CASE stControl.nTargetApplicationMode OF
	E_SEW_MoviC_Position_OperationMode.Jog:
		_bOpModeValid := TRUE;
	E_SEW_MoviC_Position_OperationMode.JogNoEnc:
		_bOpModeValid := TRUE;
	E_SEW_MoviC_Position_OperationMode.SpeedControl:
		_bOpModeValid := TRUE;
	E_SEW_MoviC_Position_OperationMode.ReferenceParam:
		_bOpModeValid := TRUE;
	E_SEW_MoviC_Position_OperationMode.ReferenceBus:
		_bOpModeValid := TRUE;
	E_SEW_MoviC_Position_OperationMode.PositionAbs, E_SEW_MoviC_Position_OperationMode.EnergyOptimized, E_SEW_MoviC_Position_OperationMode.MechanicsOptimized:
		_bOpModeValid := TRUE;
	E_SEW_MoviC_Position_OperationMode.PositionRel:
		_bOpModeValid := TRUE;
	E_SEW_MoviC_Position_OperationMode.PositionModPos:
		_bOpModeValid := TRUE;
	E_SEW_MoviC_Position_OperationMode.PositionModNeg:
		_bOpModeValid := TRUE;
	E_SEW_MoviC_Position_OperationMode.PositionModShort:
		_bOpModeValid := TRUE;
END_CASE

(* Base state of the controller *)
_fbBaseState.bStandstill := OC_Core.F_Compare(_fbBasicDrive.fVelocity, 0, 1E-3);
_fbBaseState.nControl.b0_On := stControl.b1_EnableBusStop AND _fbBaseState.eState <> E_ProfidriveGSM_State.S1_SwitchingOnInhibited;
_fbBaseState.nControl.b1_CoastStop := NOT stControl.b13_ActivateInhibit AND bSTO;
_fbBaseState.nControl.b2_QuickStop := stControl.b0_EnableEStop;
_fbBaseState.nControl.b3_EnableOperation := stControl.b7_StartStop AND _bOpModeValid;

_fbBaseState();
		
(* Set parameter of basic drive *)
IF stControl.b12_DisableSoftwareLimits THEN
	_fbBasicDrive.fPositionLimitMin := -2147483648.0;
	_fbBasicDrive.fPositionLimitMax := 2147483647.0;
	_fbBasicDrive.fTolerance := 0.1;
ELSE
	_fbBasicDrive.fPositionLimitMin := DINT_TO_REAL(stConfig.nSoftwareLimitMin);
	_fbBasicDrive.fPositionLimitMax := DINT_TO_REAL(stConfig.nSoftwareLimitMax);
	_fbBasicDrive.fTolerance := 0.1;
END_IF
					
(* Evaluate base state *)
CASE _fbBaseState.eState OF
	
(* S1, S2 or S3 -> Drive coasts to a stop or brake is applied *)
	E_ProfidriveGSM_State.S1_SwitchingOnInhibited,
	E_ProfidriveGSM_State.S2_ReadyForSwitchingOn,
	E_ProfidriveGSM_State.S3_SwitchedOn:
		_fbBasicDrive.Stop(stConfig.fDecCoastStop);

(* S4 -> Evaluate operation mode *)
	E_ProfidriveGSM_State.S4_Operation:
		Operation();

(* S5a -> Drive decelerates with application limit *)
	E_ProfidriveGSM_State.S51_RampStop:
		_fbBasicDrive.Stop(stConfig.fDecelerationLimit);
		
(* S5b -> Drive decelerates with emergency stop ramp *)
	E_ProfidriveGSM_State.S52_QuickStop:
	    _fbBasicDrive.Stop(stConfig.fDecEstop);
END_CASE
	
(* Status Word *)
stStatus.b0_InverterReady				:= TRUE;
stStatus.b1_STOInactive					:= bSTO;
stStatus.b2_PowerStageOn				:= stControl.b13_ActivateInhibit;
stStatus.b3_BrakeReleased				:= stControl.b1_EnableBusStop OR stControl.b3_ReleaseBrake;
stStatus.b4_MotorTurning				:= NOT _fbBaseState.bStandstill;
stStatus.b5_DriveReferenced				:= TRUE;
stStatus.b6_SetpointsActive		 		:= FALSE;
stStatus.b7_TargetpositionReached		:= _fbBasicDrive.bIsPositionReached;	
stStatus.b8_ErrorActive					:= FALSE;
stStatus.b9_WarningActive				:= FALSE;
stStatus.b10_DriveTrain2Active			:= stControl.b10_ActivateDriveTrain2;
stStatus.b11_SpeedSetpointReached		:= _fbBasicDrive.bIsMoving;
stStatus.b12_SoftwareLimitsDisabled		:= stControl.b12_DisableSoftwareLimits;
stStatus.b13_OutputStageInhibit			:= _fbBaseState.nStatus.b6_SwitchingOnInhibited;
stStatus.b14_StandByModeActive			:= stControl.b14_ActivateStandByMode;
stStatus.b15_MovikitHeartbeat			:= stControl.b15_MovikitHeartbeat;

(* Status values *)
stStatus.nActualSpeed := REAL_TO_INT(_fbBasicDrive.fVelocity / stConfig.fRatioVelocity);
stStatus.nActualStatus := 0;
stStatus.nActualTorque := 0;
stStatus.nDigitalInputs := nDigitalInputs;
IF _bOpModeValid THEN
	stStatus.nActualApplicationMode := stControl.nTargetApplicationMode;
END_IF
stStatus.nActualPosition := REAL_TO_DINT(_fbBasicDrive.fPosition);
	
(* Position output *)
THIS^.ControlData := _fbBasicDrive.fPosition * stConfig.fRatioPosition + stConfig.fPositionOffset;
fValue := ControlData;
END_METHOD

METHOD INTERNAL GetControlData : BOOL
IF pControl <= 0 OR stConfig.bForceMode THEN RETURN; END_IF

(* PO1 Control Word *)
F_Memcpy(ADR(stControl), pControl, 2, stConfig.bSwapProcessData);
(* PO2 Setpoint Speed *)
F_Memcpy(ADR(stControl) + 2, pControl + 2, 2, stConfig.bSwapProcessData);
(* PO3 Setpoint Acceleration *)
F_Memcpy(ADR(stControl) + 4, pControl + 4, 2, stConfig.bSwapProcessData);
(* PO4 Setpoint Deceleration *)
F_Memcpy(ADR(stControl) + 6, pControl + 6, 2, stConfig.bSwapProcessData);
(* PO5 Digital Outputs *)
F_Memcpy(ADR(stControl) + 8, pControl + 8, 2, stConfig.bSwapProcessData);
(* PO6 Target Application Mode *)
F_Memcpy(ADR(stControl) + 10, pControl + 10, 2, stConfig.bSwapProcessData);
(* PO7,PO8 Target Position *)
F_Memcpy(ADR(stControl) + 12, pControl + 12, 4, stConfig.bSwapProcessData);
END_METHOD

METHOD INTERNAL InitRun
VAR_INST
	bInitRun : BOOL := TRUE;
END_VAR
IF NOT bInitRun THEN RETURN; END_IF
bInitRun := FALSE;

IF pControl = 0 OR pStatus = 0 THEN
	ADSLOGSTR(ADSLOG_MSGTYPE_WARN, CONCAT(_sPath, ': %s'), 'Plc address not set.');
END_IF

_fbBasicDrive.fPosition := stConfig.fInitPosition;
END_METHOD

METHOD PRIVATE Operation
VAR_INST
	fTargetPos			: REAL;
	fSetpointVel		: REAL;
	fSetpointAcc		: REAL;
	fSetpointDec		: REAL;
END_VAR
(* Copy setpoint values *)
fTargetPos 		:= DINT_TO_REAL(stControl.nTargetPosition);
fSetpointVel 	:= stControl.nSetpointSpeed * stConfig.fRatioVelocity; 
fSetpointAcc 	:= stControl.nSetpointAcceleration * stConfig.fRatioAccDec;
fSetpointDec 	:= stControl.nSetpointDeceleration * stConfig.fRatioAccDec;

(* Operation statemachine *)
CASE stStatus.nActualApplicationMode OF	
	E_SEW_MoviC_Position_OperationMode.Jog:
		IF stControl.b4_JoggingCW AND NOT stControl.b5_JoggingCCW THEN
			_fbBasicDrive.MoveAbsolute(DINT_TO_REAL(stConfig.nSoftwareLimitMax), fSetpointVel, fSetpointAcc, fSetpointDec);
		ELSIF stControl.b5_JoggingCCW AND NOT stControl.b4_JoggingCW THEN
			_fbBasicDrive.MoveAbsolute(DINT_TO_REAL(stConfig.nSoftwareLimitMin), fSetpointVel, fSetpointAcc, fSetpointDec);
		ELSE
			_fbBasicDrive.Stop(fSetpointDec);
		END_IF
		
	E_SEW_MoviC_Position_OperationMode.JogNoEnc:			
		IF stControl.b4_JoggingCW AND NOT stControl.b5_JoggingCCW THEN
			_fbBasicDrive.MoveVelocity(fSetpointVel, fSetpointAcc, fSetpointDec);
		ELSIF stControl.b5_JoggingCCW AND NOT stControl.b4_JoggingCW THEN
			_fbBasicDrive.MoveVelocity(-fSetpointVel, fSetpointAcc, fSetpointDec);
		ELSE
			_fbBasicDrive.Stop(fSetpointDec);
		END_IF
		
	E_SEW_MoviC_Position_OperationMode.SpeedControl:
		_fbBasicDrive.MoveVelocity(fSetpointVel, fSetpointAcc, fSetpointDec);
	
	E_SEW_MoviC_Position_OperationMode.ReferenceParam:
		//not yet implemented
		
	E_SEW_MoviC_Position_OperationMode.ReferenceBus:
		//not yet implemented
	
	E_SEW_MoviC_Position_OperationMode.PositionAbs, E_SEW_MoviC_Position_OperationMode.EnergyOptimized, E_SEW_MoviC_Position_OperationMode.MechanicsOptimized:
		IF stControl.b7_StartStop THEN						
			_fbBasicDrive.MoveAbsolute(fTargetPos, fSetpointVel, fSetpointAcc, fSetpointDec);
		ELSE
			_fbBasicDrive.Stop(fSetpointDec);
		END_IF
	
	E_SEW_MoviC_Position_OperationMode.PositionRel:
		//not yet implemented
		
	E_SEW_MoviC_Position_OperationMode.PositionModPos:
		//not yet implemented
		
	E_SEW_MoviC_Position_OperationMode.PositionModNeg:
		//not yet implemented
		
	E_SEW_MoviC_Position_OperationMode.PositionModShort:
		//not yet implemented
END_CASE
END_METHOD

METHOD INTERNAL Safety
VAR_INPUT
END_VAR
(* Check if Movisafe is available *)
IF iMovisafe <> 0 THEN
	bSTO := iMovisafe.bSTO;
END_IF
END_METHOD

METHOD INTERNAL SetStatusData
IF pStatus <= 0 THEN RETURN; END_IF

(* PI1 Status Word *)
F_Memcpy(pStatus, ADR(stStatus), 2, stConfig.bSwapProcessData);
(* PI2 Actual Speed *)
F_Memcpy(pStatus + 2, ADR(stStatus) + 2, 2, stConfig.bSwapProcessData);
(* PI3 Actual Status *)
F_Memcpy(pStatus + 4, ADR(stStatus) + 4, 2, stConfig.bSwapProcessData);
(* PI4 Actual Torque *)
F_Memcpy(pStatus + 6, ADR(stStatus) + 6, 2, stConfig.bSwapProcessData);
(* PI5 Digital Inputs *)
F_Memcpy(pStatus + 8, ADR(stStatus) + 8, 2, stConfig.bSwapProcessData);
(* PI6 Actual Application Mode *)
F_Memcpy(pStatus + 10, ADR(stStatus) + 10, 2, stConfig.bSwapProcessData);
(* PI7,PI8 Actual Position *)
F_Memcpy(pStatus + 12, ADR(stStatus) + 12, 4, stConfig.bSwapProcessData);
END_METHOD

END_FUNCTION_BLOCK

// ---- Tests/Helpers/FB_SEW_Movisafe.TcPOU
FUNCTION_BLOCK FB_SEW_Movisafe IMPLEMENTS I_SEW_Movisafe
VAR_INPUT
	bSetSTO : BOOL;
END_VAR
VAR_OUTPUT
END_VAR
VAR
END_VAR

PROPERTY bSTO : BOOL
GET
bSTO := bSetSTO;
END_GET
END_PROPERTY

END_FUNCTION_BLOCK

// ---- Tests/Devices/FB_SEW_MoviC_Velocity_Test.TcPOU
FUNCTION_BLOCK FB_SEW_MoviC_Velocity_Test EXTENDS TcUnit.FB_TestSuite

Test_ProcessDataControl();
Test_ProcessDataStatus();
Test_Safety();
Test_Cycle_Status_Const_Mirror();
Test_Cycle_Status_Movement('Test Movement 0',0,1,FALSE,FALSE );
Test_Cycle_Status_Movement('Test Movement 1000, Gear 1',1000,1,TRUE,TRUE );
Test_Cycle_Status_Movement('Test Movement -5000, Gear 1',-5000,1,TRUE,TRUE );
Test_Cycle_Status_Movement('Test Movement 1000, Gear 5',1000,5,TRUE,TRUE );
Test_Cycle_Status_Movement('Test Movement 1000, Gear -0,5',1000,-0.5,TRUE,TRUE );

METHOD Test_Cycle_Status_Const_Mirror : REFERENCE TO FB_Test
VAR
	fbDrive 			: FB_SEW_MoviC_Velocity;
	bExpected			: BOOL;
	nIntExpected		: INT;
	nWordExpected		: WORD;
	stExpected			: ST_SEW_MoviC_Velocity_Status;
	bResult 			: BOOL;	
	nIntResult 			: INT;	
	nWordResult 		: WORD;	
	stResult			: ST_SEW_MoviC_Velocity_Status;
	
	stSetControl		: ST_SEW_MoviC_Velocity_Control;
END_VAR
TEST('Status CONST TRUE');

bExpected := TRUE;

fbDrive.Cycle();

stResult := fbDrive.stStatus;

bResult := BIT_TO_BOOL(stResult.b0_InverterReady);

AssertEquals(Expected := bExpected,
             Actual := bResult,
             Message := 'InverterReady not set correctly');

bResult := BIT_TO_BOOL(stResult.b5_DriveReferenced);
			 
AssertEquals(Expected := bExpected,
             Actual := bResult,
             Message := 'DriveReferenced not set correctly');
			 
bResult := BIT_TO_BOOL(stResult.b2_PowerStageOn);
			 
AssertEquals(Expected := bExpected,
             Actual := bResult,
             Message := 'PowerStageOn not set correctly');
	 
TEST_FINISHED();

TEST('Status CONST FALSE');

bExpected := FALSE;

fbDrive.Cycle();

stResult := fbDrive.stStatus;

bResult := BIT_TO_BOOL(stResult.b6_SetpointsActive);

AssertEquals(Expected := bExpected,
             Actual := bResult,
             Message := 'SetpointsActive not set correctly');
			 
bResult := BIT_TO_BOOL(stResult.b7_TargetpositionReached);

AssertEquals(Expected := bExpected,
             Actual := bResult,
             Message := 'TargetpositionReached not set correctly');

bResult := BIT_TO_BOOL(stResult.b8_ErrorActive);
			 
AssertEquals(Expected := bExpected,
             Actual := bResult,
             Message := 'ErrorActive not set correctly');

bResult := BIT_TO_BOOL(stResult.b9_WarningActive);
			 
AssertEquals(Expected := bExpected,
             Actual := bResult,
             Message := 'WarningActive not set correctly');
	 
TEST_FINISHED();

TEST('Status CONST 0');

nWordExpected := 0;
nIntExpected := 0;

fbDrive.Cycle();

stResult := fbDrive.stStatus;

nWordResult := stResult.nActualStatus;

AssertEquals(Expected := nWordExpected,
             Actual := nWordResult,
             Message := 'ActualStatus not set correctly');

nIntResult := stResult.nActualTorque;
			 
AssertEquals(Expected := nIntExpected,
             Actual := nIntResult,
             Message := 'ActualTorque not set correctly');
			 
nWordResult := stResult.nDigitalInputs;

AssertEquals(Expected := nWordExpected,
             Actual := nWordResult,
             Message := 'DigitalInputs not set correctly');
	 
TEST_FINISHED();


TEST('Status Mirror Control FALSE');

bExpected := FALSE;

stSetControl.b13_ActivateInhibit := bExpected;
stSetControl.b10_ActivateDriveTrain2 := bExpected;
stSetControl.b12_DisableSoftwareLimits := bExpected;
stSetControl.b14_ActivateStandByMode := bExpected;
stSetControl.b15_MovikitHeartbeat := bExpected;

fbDrive.stControl := stSetControl;

fbDrive.Cycle();

stResult := fbDrive.stStatus;

bResult := BIT_TO_BOOL(stResult.b10_DriveTrain2Active);
			 
AssertEquals(Expected := bExpected,
             Actual := bResult,
             Message := 'riveTrain2Active not set correctly');

bResult := BIT_TO_BOOL(stResult.b12_SoftwareLimitsDisabled);
			 
AssertEquals(Expected := bExpected,
             Actual := bResult,
             Message := 'SoftwareLimitsDisabled not set correctly');
			 
 bResult := BIT_TO_BOOL(stResult.b14_StandByModeActive);
			 
AssertEquals(Expected := bExpected,
             Actual := bResult,
             Message := 'StandByModeActive not set correctly');
			 
bResult := BIT_TO_BOOL(stResult.b15_MovikitHeartbeat);
			 
AssertEquals(Expected := bExpected,
             Actual := bResult,
             Message := 'MovikitHeartbeat not set correctly');
	 
TEST_FINISHED();

TEST('Status Mirror Control TRUE');

bExpected := TRUE;

stSetControl.b13_ActivateInhibit := bExpected;
stSetControl.b10_ActivateDriveTrain2 := bExpected;
stSetControl.b12_DisableSoftwareLimits := bExpected;
stSetControl.b14_ActivateStandByMode := bExpected;
stSetControl.b15_MovikitHeartbeat := bExpected;

fbDrive.stControl := stSetControl;

fbDrive.Cycle();

stResult := fbDrive.stStatus;

bResult := BIT_TO_BOOL(stResult.b10_DriveTrain2Active);
			 
AssertEquals(Expected := bExpected,
             Actual := bResult,
             Message := 'DriveTrain2Active not set correctly');

bResult := BIT_TO_BOOL(stResult.b12_SoftwareLimitsDisabled);
			 
AssertEquals(Expected := bExpected,
             Actual := bResult,
             Message := 'SoftwareLimitsDisabled not set correctly');
			 
 bResult := BIT_TO_BOOL(stResult.b14_StandByModeActive);
			 
AssertEquals(Expected := bExpected,
             Actual := bResult,
             Message := 'StandByModeActive not set correctly');
			 
bResult := BIT_TO_BOOL(stResult.b15_MovikitHeartbeat);
			 
AssertEquals(Expected := bExpected,
             Actual := bResult,
             Message := 'MovikitHeartbeat not set correctly');
	 
TEST_FINISHED();
END_METHOD

METHOD Test_Cycle_Status_Movement : REFERENCE TO FB_Test
VAR_INPUT
	sName 								: T_MaxString;
	nVelcity							: INT;
	fRatioVelcity						: REAL;
	bExpected_b4_MotorTurning 			: BOOL;
	bExpected_b11_SpeedSetpointReached 	: BOOL;
END_VAR
VAR
	nCycle		: INT;
	fbDrive 	: FB_SEW_MoviC_Velocity;
	bResult		: BOOL;	
	nResult 	: INT;
END_VAR
TEST(sName);

// Start Conditions
fbDrive.stControl.b0_EnableEStop := TRUE;
fbDrive.stControl.b1_EnableBusStop := TRUE;
fbDrive.stControl.b7_StartStop := TRUE;
fbDrive.stControl.b13_ActivateInhibit := FALSE;
fbDrive.bSTO := TRUE;
fbDrive.stControl.nSetpointSpeed := nVelcity;
fbDrive.stControl.nSetpointAcceleration := 1000;
fbDrive.stControl.nSetpointDeceleration := 1000;

fbDrive.stConfig.fRatioPosition := fRatioVelcity;

FOR nCycle := 1 TO 5500 DO
	fbDrive.Cycle();
END_FOR

nResult := fbDrive.stStatus.nActualSpeed;

AssertEquals(Expected := nVelcity,
             Actual := nResult,
             Message := 'ActualSpeed not set correctly');

bResult := fbDrive.stStatus.b4_MotorTurning;

AssertEquals(Expected := bExpected_b4_MotorTurning,
             Actual := bResult,
             Message := 'b4_MotorTurning not set correctly');


bResult := fbDrive.stStatus.b11_SpeedSetpointReached;
			 
AssertEquals(Expected := bExpected_b11_SpeedSetpointReached,
             Actual := bResult,
             Message := 'b11_SpeedSetpointReached not set correctly');
	 
TEST_FINISHED();
END_METHOD

METHOD Test_ProcessDataControl : REFERENCE TO FB_Test
VAR
	fbDrive 						: FB_SEW_MoviC_Velocity;
	
	nExpectedCW						: WORD;
	nExpectedSetpointSpeed			: INT;
	nExpectedSetpointAcceleration	: INT;
	nExpectedSetpointDeceleration	: INT;
	nExpectedDigitalOutputs			: WORD;
	
	nActualCW						: WORD;
	nActualSetpointSpeed			: INT;
	nActualSetpointAcceleration		: INT;
	nActualSetpointDeceleration		: INT;
	nActualDigitalOutputs			: WORD;
		
	stExpectedControlData 			: ST_SEW_MoviC_Velocity_Control;		
	stActualControlData				: ST_SEW_MoviC_Velocity_Control;	
END_VAR
TEST('Process data to control structure');

//Arrange
nExpectedCW := 16#A1B2;					
nExpectedSetpointSpeed := UINT_TO_INT(16#C3D4);		
nExpectedSetpointAcceleration := UINT_TO_INT(16#E5F6);		
nExpectedSetpointDeceleration := UINT_TO_INT(16#B6A5);	
nExpectedDigitalOutputs := 16#D4C3;			

F_Memcpy(ADR(stExpectedControlData), ADR(nExpectedCW), 2, FALSE);
F_Memcpy(ADR(stExpectedControlData) + 2, ADR(nExpectedSetpointSpeed), 2, FALSE);
F_Memcpy(ADR(stExpectedControlData) + 4, ADR(nExpectedSetpointAcceleration), 2, FALSE);
F_Memcpy(ADR(stExpectedControlData) + 6, ADR(nExpectedSetpointDeceleration), 2, FALSE);
F_Memcpy(ADR(stExpectedControlData) + 8, ADR(nExpectedDigitalOutputs), 2, FALSE);

fbDrive.pControl := ADR(stExpectedControlData);

//Act
fbDrive.GetControlData();

stActualControlData := fbDrive.stControl;

//Assert
F_Memcpy(ADR(nActualCW), ADR(fbDrive.stControl), 2, FALSE);
//F_Memcpy(ADR(nActualTargetVelocity), ADR(fbDrive.stControl) + 2, 2, FALSE);

AssertEquals(Expected := nExpectedCW,
             Actual := nActualCW,
             Message := 'CW is not correct');
	 
AssertEquals(Expected := nExpectedSetpointSpeed,
             Actual := stActualControlData.nSetpointSpeed,
             Message := 'SetpointSpeed is not correct');
			 
AssertEquals(Expected := nExpectedSetpointAcceleration,
             Actual := stActualControlData.nSetpointAcceleration,
             Message := 'SetpointAcceleration is not correct');
			 
AssertEquals(Expected := nExpectedSetpointDeceleration,
             Actual := stActualControlData.nSetpointDeceleration,
             Message := 'SetpointSpeed is not correct');
			 
AssertEquals(Expected := nExpectedDigitalOutputs,
             Actual := stActualControlData.nDigitalOutputs,
             Message := 'SetpointDeceleration is not correct');
			 
TEST_FINISHED();


TEST('Process data to control structure SWAP');

//Arrange
F_Memcpy(ADR(stExpectedControlData), ADR(nExpectedCW), 2, TRUE);
F_Memcpy(ADR(stExpectedControlData) + 2, ADR(nExpectedSetpointSpeed), 2, TRUE);
F_Memcpy(ADR(stExpectedControlData) + 4, ADR(nExpectedSetpointAcceleration), 2, TRUE);
F_Memcpy(ADR(stExpectedControlData) + 6, ADR(nExpectedSetpointDeceleration), 2, TRUE);
F_Memcpy(ADR(stExpectedControlData) + 8, ADR(nExpectedDigitalOutputs), 2, TRUE);

fbDrive.stConfig.bSwapProcessData := TRUE;

fbDrive.pControl := ADR(stExpectedControlData);

//Act
fbDrive.GetControlData();

stActualControlData := fbDrive.stControl;

//Assert
AssertEquals(Expected := nExpectedCW,
             Actual := nActualCW,
             Message := 'CW is not correct');
	 
AssertEquals(Expected := nExpectedSetpointSpeed,
             Actual := stActualControlData.nSetpointSpeed,
             Message := 'SetpointSpeed is not correct');
			 
AssertEquals(Expected := nExpectedSetpointAcceleration,
             Actual := stActualControlData.nSetpointAcceleration,
             Message := 'SetpointAcceleration is not correct');
			 
AssertEquals(Expected := nExpectedSetpointDeceleration,
             Actual := stActualControlData.nSetpointDeceleration,
             Message := 'SetpointSpeed is not correct');
			 
AssertEquals(Expected := nExpectedDigitalOutputs,
             Actual := stActualControlData.nDigitalOutputs,
             Message := 'SetpointDeceleration is not correct');

TEST_FINISHED();
END_METHOD

METHOD Test_ProcessDataStatus : REFERENCE TO FB_Test
VAR
	fbDrive 						: FB_SEW_MoviC_Velocity;
	
	nExpectedSW						: WORD;
	nExpectedActualSpeed			: INT;
	nExpectedActualStatus			: WORD;
	nExpectedActualTorque			: INT;
	nExpectedDigitalInputs			: WORD;
	
	nActualSW						: WORD;
	nActualActualSpeed				: INT;
	nActualActualStatus				: WORD;
	nActualActualTorque				: INT;
	nActualDigitalInputs			: WORD;

	stExpectedStatusData 			: ST_SEW_MoviC_Velocity_Status;		
	stActualStatusData 				: ST_SEW_MoviC_Velocity_Status;	
END_VAR
TEST('Assign status structure to process data');

//Arrange
nExpectedSW := 16#A1B2;					
nExpectedActualSpeed := UINT_TO_INT(16#C3D4);		
nExpectedActualStatus := 16#E5F6;		
nExpectedActualTorque := UINT_TO_INT(16#B6A5);	
nExpectedDigitalInputs := 16#B6A5;			
	
F_Memcpy(ADR(fbDrive.stStatus), ADR(nExpectedSW), 2, FALSE);
F_Memcpy(ADR(fbDrive.stStatus) + 2, ADR(nExpectedActualSpeed), 2, FALSE);
F_Memcpy(ADR(fbDrive.stStatus) + 4, ADR(nExpectedActualStatus), 2, FALSE);
F_Memcpy(ADR(fbDrive.stStatus) + 6, ADR(nExpectedActualTorque), 2, FALSE);
F_Memcpy(ADR(fbDrive.stStatus) + 8, ADR(nExpectedDigitalInputs), 2, FALSE);

fbDrive.pStatus := ADR(stActualStatusData);

//Act
fbDrive.SetStatusData();

//Assert
F_Memcpy(ADR(nActualSW), ADR(stActualStatusData), 2, FALSE);
F_Memcpy(ADR(nActualActualSpeed), ADR(stActualStatusData) + 2, 2, FALSE);
F_Memcpy(ADR(nActualActualStatus), ADR(stActualStatusData) + 4, 2, FALSE);
F_Memcpy(ADR(nActualActualTorque), ADR(stActualStatusData) + 6, 2, FALSE);
F_Memcpy(ADR(nActualDigitalInputs), ADR(stActualStatusData) + 8, 2, FALSE);

AssertEquals(Expected := nExpectedSW,
             Actual := nActualSW,
             Message := 'ZSW1 is not correct');
	 
AssertEquals(Expected := nExpectedActualSpeed,
             Actual := nActualActualSpeed,
             Message := 'ActualVelocity is not correct');	

AssertEquals(Expected := nExpectedActualStatus,
             Actual := nActualActualStatus,
             Message := 'ActualVelocity is not correct');

AssertEquals(Expected := nExpectedActualTorque,
             Actual := nActualActualTorque,
             Message := 'ActualVelocity is not correct');	
				 
AssertEquals(Expected := nExpectedDigitalInputs,
             Actual := nActualDigitalInputs,
             Message := 'ActualVelocity is not correct');	
					 			 
TEST_FINISHED();

TEST('Assign status structure to process data SWAP');

//Arrange
nExpectedSW := 16#A1B2;					
nExpectedActualSpeed := UINT_TO_INT(16#C3D4);		
nExpectedActualStatus := 16#E5F6;		
nExpectedActualTorque := UINT_TO_INT(16#B6A5);	
nExpectedDigitalInputs := 16#B6A5;			
	
F_Memcpy(ADR(fbDrive.stStatus), ADR(nExpectedSW), 2, TRUE);
F_Memcpy(ADR(fbDrive.stStatus) + 2, ADR(nExpectedActualSpeed), 2, TRUE);
F_Memcpy(ADR(fbDrive.stStatus) + 4, ADR(nExpectedActualStatus), 2, TRUE);
F_Memcpy(ADR(fbDrive.stStatus) + 6, ADR(nExpectedActualTorque), 2, TRUE);
F_Memcpy(ADR(fbDrive.stStatus) + 8, ADR(nExpectedDigitalInputs), 2, TRUE);

fbDrive.stConfig.bSwapProcessData := TRUE;

fbDrive.pStatus := ADR(stActualStatusData);

//Act
fbDrive.SetStatusData();

//Assert
F_Memcpy(ADR(nActualSW), ADR(stActualStatusData), 2, FALSE);
F_Memcpy(ADR(nActualActualSpeed), ADR(stActualStatusData) + 2, 2, FALSE);
F_Memcpy(ADR(nActualActualStatus), ADR(stActualStatusData) + 4, 2, FALSE);
F_Memcpy(ADR(nActualActualTorque), ADR(stActualStatusData) + 6, 2, FALSE);
F_Memcpy(ADR(nActualDigitalInputs), ADR(stActualStatusData) + 8, 2, FALSE);

AssertEquals(Expected := nExpectedSW,
             Actual := nActualSW,
             Message := 'ZSW1 is not correct');
	 
AssertEquals(Expected := nExpectedActualSpeed,
             Actual := nActualActualSpeed,
             Message := 'ActualVelocity is not correct');	

AssertEquals(Expected := nExpectedActualStatus,
             Actual := nActualActualStatus,
             Message := 'ActualVelocity is not correct');

AssertEquals(Expected := nExpectedActualTorque,
             Actual := nActualActualTorque,
             Message := 'ActualVelocity is not correct');	
				 
AssertEquals(Expected := nExpectedDigitalInputs,
             Actual := nActualDigitalInputs,
             Message := 'ActualVelocity is not correct');			 
			 
TEST_FINISHED();
END_METHOD

METHOD Test_Safety : REFERENCE TO FB_Test
VAR
	fbDrive 					: FB_SEW_MoviC_Velocity;
		
	fbSafe						: FB_SEW_Movisafe;
	
	stExpectedSTO				: BOOL;		
	stActualSTO					: BOOL;	
END_VAR
TEST(' Without Safety Interface STO TRUE');

//Arrange
stExpectedSTO := TRUE;
fbDrive.bSTO := stExpectedSTO;

//Act
fbDrive.Safety();

//Assert
stActualSTO := fbDrive.bSTO;

AssertEquals(Expected := stExpectedSTO,
             Actual := stActualSTO,
             Message := 'STO is not correct');
	 		 
TEST_FINISHED();

TEST(' Without Safety Interface STO FALSE');

//Arrange
stExpectedSTO := FALSE;
fbDrive.bSTO := stExpectedSTO;

//Act
fbDrive.Safety();

//Assert
stActualSTO := fbDrive.bSTO;

AssertEquals(Expected := stExpectedSTO,
             Actual := stActualSTO,
             Message := 'STO is not correct');
	 		 
TEST_FINISHED();

TEST('Safety Interface STO TRUE');

//Arrange
stExpectedSTO := TRUE;

fbSafe.bSetSTO := stExpectedSTO;
fbDrive.iMovisafe := fbSafe;

//Act
fbDrive.Safety();

//Assert
stActualSTO := fbDrive.bSTO;

AssertEquals(Expected := stExpectedSTO,
             Actual := stActualSTO,
             Message := 'STO is not correct');
	 		 
TEST_FINISHED();

TEST('Safety Interface FALSE');

//Arrange
stExpectedSTO := FALSE;

fbSafe.bSetSTO := stExpectedSTO;
fbDrive.iMovisafe := fbSafe;

//Act
fbDrive.Safety();

//Assert
stActualSTO := fbDrive.bSTO;

AssertEquals(Expected := stExpectedSTO,
             Actual := stActualSTO,
             Message := 'STO is not correct');
	 		 
TEST_FINISHED();

TEST('Safety Interface false, Overwrite FB input');

//Arrange
stExpectedSTO := FALSE;

fbSafe.bSetSTO := stExpectedSTO;
fbDrive.iMovisafe := fbSafe;
fbDrive.bSTO := NOT stExpectedSTO;

//Act
fbDrive.Safety();

//Assert
stActualSTO := fbDrive.bSTO;

AssertEquals(Expected := stExpectedSTO,
             Actual := stActualSTO,
             Message := 'STO is not correct');
	 		 
TEST_FINISHED();

TEST('Safety Interface true, Overwrite FB input');

//Arrange
stExpectedSTO := TRUE;

fbSafe.bSetSTO := stExpectedSTO;
fbDrive.iMovisafe := fbSafe;
fbDrive.bSTO := NOT stExpectedSTO;

//Act
fbDrive.Safety();

//Assert
stActualSTO := fbDrive.bSTO;

AssertEquals(Expected := stExpectedSTO,
             Actual := stActualSTO,
             Message := 'STO is not correct');
	 		 
TEST_FINISHED();
END_METHOD

END_FUNCTION_BLOCK

// ---- Devices/SEW_MoviC_Velocity/FB_SEW_MoviC_Velocity.TcPOU
(*
FB_SEW_MoviC_Velocity simulates the funcitionalty of a SEW‑EURODRIVE MOVI-C® CONTROLLER with MOVIKIT® Velocity module.

Disclaimer: This simulation is an independent project and is not affiliated with, endorsed by, or approved by SEW‑EURODRIVE. All rights to the SEW‑EURODRIVE brand name and trademarks remain the property of the manufacturer.
Furthermore, no guarantee is given for the completeness of the functional scope or the error-free operation of the simulation. Users should be aware that deviations from the actual product may occur.
*)

{attribute 'reflection'}
FUNCTION_BLOCK FB_SEW_MoviC_Velocity EXTENDS FB_LinkDataReal

VAR_INPUT
	pControl 			: PVOID; //Pocess data from fieldbus. Size must be >= stControl.
	pStatus 			: PVOID; //Pocess data to fieldbus. Size must be >= stStatus.
	stControl 			: ST_SEW_MoviC_Velocity_Control; //Control structure. Is read from the fieldbus.
	stConfig 			: ST_SEW_MoviC_Velocity_Config; //Config structure. Contains parameters of the device.	
	
	bSTO				: BOOL := TRUE;
	iMovisafe			: I_SEW_Movisafe;
END_VAR

VAR_OUTPUT
	stStatus			: ST_SEW_MoviC_Velocity_Status;
	fValue				: REAL;
END_VAR

VAR
    {attribute 'instance-path'} 
    {attribute 'noinit'} 
    _sPath 				: STRING; 	                			
	                			
	_fbBaseState		: FB_ProfidriveGSM;
	_fbBasicDrive		: FB_DriveControl;	                						
END_VAR

SUPER^();
InitRun();

GetControlData();
Safety();
Cycle();
SetStatusData();

METHOD INTERNAL Cycle
(* Base state of the controller *)
_fbBaseState.bStandstill := OC_Core.F_Compare(_fbBasicDrive.fVelocity, 0, 1E-3);
_fbBaseState.nControl.b0_On := stControl.b1_EnableBusStop AND _fbBaseState.eState <> E_ProfidriveGSM_State.S1_SwitchingOnInhibited;
_fbBaseState.nControl.b1_CoastStop := NOT stControl.b13_ActivateInhibit AND bSTO;
_fbBaseState.nControl.b2_QuickStop := stControl.b0_EnableEStop;
_fbBaseState.nControl.b3_EnableOperation := stControl.b7_StartStop;

_fbBaseState();
					
(* Evaluate base state *)
CASE _fbBaseState.eState OF	
(* S1, S2 or S3 -> Drive coasts to a stop or brake is applied *)
	E_ProfidriveGSM_State.S1_SwitchingOnInhibited,
	E_ProfidriveGSM_State.S2_ReadyForSwitchingOn,
	E_ProfidriveGSM_State.S3_SwitchedOn:
		_fbBasicDrive.Stop(stConfig.fDecCoastStop);

(* S4 -> Operation mode *)
	E_ProfidriveGSM_State.S4_Operation:
		Operation();

(* S5a -> Drive decelerates with application limit *)
	E_ProfidriveGSM_State.S51_RampStop:
		_fbBasicDrive.Stop(stConfig.fDecelerationLimit);
		
(* S5b -> Drive decelerates with emergency stop ramp *)
	E_ProfidriveGSM_State.S52_QuickStop:
	    _fbBasicDrive.Stop(stConfig.fDecEstop);
END_CASE
	
(* Status Word *)
stStatus.b0_InverterReady				:= TRUE;
stStatus.b1_STOInactive					:= bSTO;
stStatus.b2_PowerStageOn				:= _fbBaseState.bPowerOn;
stStatus.b3_BrakeReleased				:= stControl.b1_EnableBusStop OR stControl.b3_ReleaseBrake;
stStatus.b4_MotorTurning				:= NOT _fbBaseState.bStandstill;
stStatus.b5_DriveReferenced				:= TRUE;
stStatus.b6_SetpointsActive		 		:= FALSE;
stStatus.b7_TargetpositionReached		:= FALSE;	
stStatus.b8_ErrorActive					:= FALSE;
stStatus.b9_WarningActive				:= FALSE;
stStatus.b10_DriveTrain2Active			:= stControl.b10_ActivateDriveTrain2;
stStatus.b11_SpeedSetpointReached		:= _fbBasicDrive.bIsMoving;
stStatus.b12_SoftwareLimitsDisabled		:= stControl.b12_DisableSoftwareLimits;
stStatus.b13_OutputStageInhibit			:= _fbBaseState.nStatus.b6_SwitchingOnInhibited;
stStatus.b14_StandByModeActive			:= stControl.b14_ActivateStandByMode;
stStatus.b15_MovikitHeartbeat			:= stControl.b15_MovikitHeartbeat;

(* Status values *)
stStatus.nActualSpeed := REAL_TO_INT(_fbBasicDrive.fVelocity / stConfig.fRatioVelocity);
stStatus.nActualStatus := 0;
stStatus.nActualTorque := 0;
stStatus.nDigitalInputs := 0;
	
(* Output of actual value *)	
IF stConfig.bOutputVelocity THEN
	ControlData := _fbBasicDrive.fVelocity / stConfig.fRatioVelocity;
ELSE
	ControlData := ControlData + _fbBasicDrive.fVelocity / stConfig.fRatioVelocity *  GVL_Core.fbSystem.fDeltaTime * GVL_Core.fbSystem.fTimeScaling;
END_IF

fValue := ControlData;
END_METHOD

METHOD INTERNAL GetControlData : BOOL
IF pControl <= 0 OR stConfig.bForceMode THEN RETURN; END_IF

(* PO1 Control Word *)
F_Memcpy(ADR(stControl), pControl, 2, stConfig.bSwapProcessData);
(* PO2 Setpoint Speed *)
F_Memcpy(ADR(stControl) + 2, pControl + 2, 2, stConfig.bSwapProcessData);
(* PO3 Setpoint Acceleration *)
F_Memcpy(ADR(stControl) + 4, pControl + 4, 2, stConfig.bSwapProcessData);
(* PO4 Setpoint Deceleration *)
F_Memcpy(ADR(stControl) + 6, pControl + 6, 2, stConfig.bSwapProcessData);
(* PO5 Digital Outputs *)
F_Memcpy(ADR(stControl) + 8, pControl + 8, 2, stConfig.bSwapProcessData);
END_METHOD

METHOD INTERNAL InitRun
VAR_INST
	bInitRun : BOOL := TRUE;
END_VAR
IF NOT bInitRun THEN RETURN; END_IF
bInitRun := FALSE;

IF pControl = 0 OR pStatus = 0 THEN
	ADSLOGSTR(ADSLOG_MSGTYPE_WARN, CONCAT(_sPath, ': %s'), 'Plc address not set.');
END_IF

_fbBasicDrive.fPosition := stConfig.fInitPosition;
END_METHOD

METHOD PRIVATE Operation
VAR_INST
	fTargetPos			: REAL;
	fSetpointVel		: REAL;
	fSetpointAcc		: REAL;
	fSetpointDec		: REAL;
END_VAR
(* Copy setpoint values *)
fSetpointVel 	:= stControl.nSetpointSpeed * stConfig.fRatioVelocity; 
fSetpointAcc 	:= stControl.nSetpointAcceleration * stConfig.fRatioAccDec;

_fbBasicDrive.MoveVelocity(fSetpointVel, fSetpointAcc, fSetpointAcc);
END_METHOD

METHOD INTERNAL Safety
VAR_INPUT
END_VAR
(* Check if Movisafe is available *)
IF iMovisafe <> 0 THEN
	bSTO := iMovisafe.bSTO;
END_IF
END_METHOD

METHOD INTERNAL SetStatusData
IF pStatus <= 0 THEN RETURN; END_IF

(* PI1 Status Word *)
F_Memcpy(pStatus, ADR(stStatus), 2, stConfig.bSwapProcessData);
(* PI2 Actual Speed *)
F_Memcpy(pStatus + 2, ADR(stStatus) + 2, 2, stConfig.bSwapProcessData);
(* PI3 Actual Status *)
F_Memcpy(pStatus + 4, ADR(stStatus) + 4, 2, stConfig.bSwapProcessData);
(* PI4 Actual Torque *)
F_Memcpy(pStatus + 6, ADR(stStatus) + 6, 2, stConfig.bSwapProcessData);
(* PI5 Digital Inputs *)
F_Memcpy(pStatus + 8, ADR(stStatus) + 8, 2, stConfig.bSwapProcessData);
END_METHOD

END_FUNCTION_BLOCK

// ---- Tests/Devices/FB_SEW_Movisafe_CSSx1a_Test.TcPOU
FUNCTION_BLOCK FB_SEW_Movisafe_CSSx1a_Test EXTENDS TcUnit.FB_TestSuite

Test_Cycle();
Test_ProcessDataControl();
Test_ProcessDataStatus();

METHOD Test_Cycle : REFERENCE TO FB_Test
VAR
	fbDevice 						: FB_SEW_Movisafe_CSSx1a;
	
	stSetControl					: ST_SEW_Movisafe_CSSx1a_Control;

	stExpectedStatusData 			: ST_SEW_Movisafe_CSSx1a_Status;		
	stActualStatusData 				: ST_SEW_Movisafe_CSSx1a_Status;	
END_VAR
TEST('Cycle Control FALSE');

//Arrange
stSetControl.b0_0_STO				:=	FALSE;	
stSetControl.b0_1_SLI			    :=  FALSE;
stSetControl.b0_2_SBT			    :=  FALSE;
stSetControl.b0_3_Reserved		    :=  FALSE;
stSetControl.b0_4_MutingEncErr	    :=  FALSE;
stSetControl.b0_5_TestModeActice	:=  FALSE;
stSetControl.b0_6_AckFDI			:=  FALSE;
stSetControl.b0_7_AckError		    :=  FALSE;
stSetControl.b1_0_F_DO0			    :=  FALSE;
stSetControl.b1_1_F_DO1			    :=  FALSE;
stSetControl.b1_2_Reserved		    :=  FALSE;
stSetControl.b1_3_Reserved		    :=  FALSE;
stSetControl.b1_4_Reserved		    :=  FALSE;
stSetControl.b1_5_Reserved		    :=  FALSE;
stSetControl.b1_6_Reserved		    :=  FALSE;
stSetControl.b1_7_Reserved		    :=  FALSE;
stSetControl.b2_0_SOS1			    :=  FALSE;
stSetControl.b2_1_Reserved		    :=  FALSE;
stSetControl.b2_2_SSx1			    :=  FALSE;
stSetControl.b2_3_SSx2			    :=  FALSE;
stSetControl.b2_4_SDI1			    :=  FALSE;
stSetControl.b2_5_SDI2			    :=  FALSE;
stSetControl.b2_6_SLI1			    :=  FALSE;
stSetControl.b2_7_SLI2			    :=  FALSE;
stSetControl.b3_0_SLS1			    :=  FALSE;
stSetControl.b3_1_SLS2			    :=  FALSE;
stSetControl.b3_2_SLS3			    :=  FALSE;
stSetControl.b3_3_SLS4			    :=  FALSE;
stSetControl.b3_4_SSR1			    :=  FALSE;
stSetControl.b3_5_SSR2			    :=  FALSE;
stSetControl.b3_6_Reserved		    :=  FALSE;
stSetControl.b3_7_Reserved		    :=  FALSE;
stSetControl.b4_0_SLA1			    :=  FALSE;
stSetControl.b4_1_SLA2			    :=  FALSE;
stSetControl.b4_2_Reserved		    :=  FALSE;
stSetControl.b4_3_Reserved		    :=  FALSE;
stSetControl.b4_4_Reserved		    :=  FALSE;
stSetControl.b4_5_Reserved		    :=  FALSE;
stSetControl.b4_6_Reserved		    :=  FALSE;
stSetControl.b4_7_Reserved		    :=  FALSE;

stExpectedStatusData.b0_0_STOActive			:= stSetControl.b0_0_STO;
stExpectedStatusData.b0_1_ASFDiag		    := FALSE;
stExpectedStatusData.b0_2_SBTActive		    := FALSE;
stExpectedStatusData.b0_3_InputDataValid	:= TRUE;
stExpectedStatusData.b0_4_MutingEncErr	    := stSetControl.b0_4_MutingEncErr;
stExpectedStatusData.b0_5_TestModeActive	:= stSetControl.b0_5_TestModeActice;
stExpectedStatusData.b0_6_Warning		    := FALSE;
stExpectedStatusData.b0_7_ErrorState		:= FALSE;
stExpectedStatusData.b1_0_F_DI0			    := FALSE;
stExpectedStatusData.b1_1_F_DI1			    := FALSE;
stExpectedStatusData.b1_2_F_DI2			    := FALSE;
stExpectedStatusData.b1_3_F_DI3			    := FALSE;
stExpectedStatusData.b1_4_Reserved		    := FALSE;
stExpectedStatusData.b1_5_Reserved		    := FALSE;
stExpectedStatusData.b1_6_Reserved		    := FALSE;
stExpectedStatusData.b1_7_Reserved		    := FALSE;
stExpectedStatusData.b2_0_SOS1			    := NOT stSetControl.b2_0_SOS1;
stExpectedStatusData.b2_1_Reserved		    := FALSE;                  
stExpectedStatusData.b2_2_SSx1			    := NOT stSetControl.b2_2_SSx1;
stExpectedStatusData.b2_3_SSx2			    := NOT stSetControl.b2_3_SSx2;
stExpectedStatusData.b2_4_SDI1			    := NOT stSetControl.b2_4_SDI1;
stExpectedStatusData.b2_5_SDI2			    := NOT stSetControl.b2_5_SDI2;
stExpectedStatusData.b2_6_SLI1			    := NOT stSetControl.b2_6_SLI1;
stExpectedStatusData.b2_7_SLI2			    := NOT stSetControl.b2_7_SLI2;
stExpectedStatusData.b3_0_SLS1			    := NOT stSetControl.b3_0_SLS1;
stExpectedStatusData.b3_1_SLS2			    := NOT stSetControl.b3_1_SLS2;
stExpectedStatusData.b3_2_SLS3			    := NOT stSetControl.b3_2_SLS3;
stExpectedStatusData.b3_3_SLS4			    := NOT stSetControl.b3_3_SLS4;
stExpectedStatusData.b3_4_SSR1			    := NOT stSetControl.b3_4_SSR1;
stExpectedStatusData.b3_5_SSR2			    := NOT stSetControl.b3_5_SSR2;
stExpectedStatusData.b3_6_Reserved		    := FALSE;
stExpectedStatusData.b3_7_Reserved		    := FALSE;
stExpectedStatusData.b4_0_SLA1			    := NOT stSetControl.b4_0_SLA1;
stExpectedStatusData.b4_1_SLA2			    := NOT stSetControl.b4_1_SLA2;
stExpectedStatusData.b4_2_SSM1			    := FALSE;
stExpectedStatusData.b4_3_SSM2			    := FALSE;
stExpectedStatusData.b4_4_SSM3			    := FALSE;
stExpectedStatusData.b4_5_SSM4			    := FALSE;
stExpectedStatusData.b4_6_Reserved		    := FALSE;
stExpectedStatusData.b4_7_Reserved		    := FALSE;
stExpectedStatusData.b5_0_Reserved		    := FALSE;
stExpectedStatusData.b5_1_Reserved		    := FALSE;
stExpectedStatusData.b5_2_Reserved		    := FALSE;
stExpectedStatusData.b5_3_Reserved		    := FALSE;
stExpectedStatusData.b5_4_Reserved		    := FALSE;
stExpectedStatusData.b5_5_Reserved		    := FALSE;
stExpectedStatusData.b5_6_Reserved		    := FALSE;
stExpectedStatusData.b5_7_Reserved	        := FALSE;
	
//Act

fbDevice.stControl := stSetControl;
fbDevice.Cycle();
stActualStatusData := fbDevice.stStatus ;

//Assert

AssertEquals(Expected := stExpectedStatusData,
             Actual := stActualStatusData,
             Message := 'Status is not correct');
	 					 			 
TEST_FINISHED();

TEST('Cycle Control TRUE');

//Arrange
stSetControl.b0_0_STO				:=	TRUE;	
stSetControl.b0_1_SLI			    :=  TRUE;
stSetControl.b0_2_SBT			    :=  TRUE;
stSetControl.b0_3_Reserved		    :=  TRUE;
stSetControl.b0_4_MutingEncErr	    :=  TRUE;
stSetControl.b0_5_TestModeActice	:=  TRUE;
stSetControl.b0_6_AckFDI			:=  TRUE;
stSetControl.b0_7_AckError		    :=  TRUE;
stSetControl.b1_0_F_DO0			    :=  TRUE;
stSetControl.b1_1_F_DO1			    :=  TRUE;
stSetControl.b1_2_Reserved		    :=  TRUE;
stSetControl.b1_3_Reserved		    :=  TRUE;
stSetControl.b1_4_Reserved		    :=  TRUE;
stSetControl.b1_5_Reserved		    :=  TRUE;
stSetControl.b1_6_Reserved		    :=  TRUE;
stSetControl.b1_7_Reserved		    :=  TRUE;
stSetControl.b2_0_SOS1			    :=  TRUE;
stSetControl.b2_1_Reserved		    :=  TRUE;
stSetControl.b2_2_SSx1			    :=  TRUE;
stSetControl.b2_3_SSx2			    :=  TRUE;
stSetControl.b2_4_SDI1			    :=  TRUE;
stSetControl.b2_5_SDI2			    :=  TRUE;
stSetControl.b2_6_SLI1			    :=  TRUE;
stSetControl.b2_7_SLI2			    :=  TRUE;
stSetControl.b3_0_SLS1			    :=  TRUE;
stSetControl.b3_1_SLS2			    :=  TRUE;
stSetControl.b3_2_SLS3			    :=  TRUE;
stSetControl.b3_3_SLS4			    :=  TRUE;
stSetControl.b3_4_SSR1			    :=  TRUE;
stSetControl.b3_5_SSR2			    :=  TRUE;
stSetControl.b3_6_Reserved		    :=  TRUE;
stSetControl.b3_7_Reserved		    :=  TRUE;
stSetControl.b4_0_SLA1			    :=  TRUE;
stSetControl.b4_1_SLA2			    :=  TRUE;
stSetControl.b4_2_Reserved		    :=  TRUE;
stSetControl.b4_3_Reserved		    :=  TRUE;
stSetControl.b4_4_Reserved		    :=  TRUE;
stSetControl.b4_5_Reserved		    :=  TRUE;
stSetControl.b4_6_Reserved		    :=  TRUE;
stSetControl.b4_7_Reserved		    :=  TRUE;

stExpectedStatusData.b0_0_STOActive			:= stSetControl.b0_0_STO;
stExpectedStatusData.b0_1_ASFDiag		    := FALSE;
stExpectedStatusData.b0_2_SBTActive		    := FALSE;
stExpectedStatusData.b0_3_InputDataValid	:= TRUE;
stExpectedStatusData.b0_4_MutingEncErr	    := stSetControl.b0_4_MutingEncErr;
stExpectedStatusData.b0_5_TestModeActive	:= stSetControl.b0_5_TestModeActice;
stExpectedStatusData.b0_6_Warning		    := FALSE;
stExpectedStatusData.b0_7_ErrorState		:= FALSE;
stExpectedStatusData.b1_0_F_DI0			    := FALSE;
stExpectedStatusData.b1_1_F_DI1			    := FALSE;
stExpectedStatusData.b1_2_F_DI2			    := FALSE;
stExpectedStatusData.b1_3_F_DI3			    := FALSE;
stExpectedStatusData.b1_4_Reserved		    := FALSE;
stExpectedStatusData.b1_5_Reserved		    := FALSE;
stExpectedStatusData.b1_6_Reserved		    := FALSE;
stExpectedStatusData.b1_7_Reserved		    := FALSE;
stExpectedStatusData.b2_0_SOS1			    := NOT stSetControl.b2_0_SOS1;
stExpectedStatusData.b2_1_Reserved		    := FALSE;                  
stExpectedStatusData.b2_2_SSx1			    := NOT stSetControl.b2_2_SSx1;
stExpectedStatusData.b2_3_SSx2			    := NOT stSetControl.b2_3_SSx2;
stExpectedStatusData.b2_4_SDI1			    := NOT stSetControl.b2_4_SDI1;
stExpectedStatusData.b2_5_SDI2			    := NOT stSetControl.b2_5_SDI2;
stExpectedStatusData.b2_6_SLI1			    := NOT stSetControl.b2_6_SLI1;
stExpectedStatusData.b2_7_SLI2			    := NOT stSetControl.b2_7_SLI2;
stExpectedStatusData.b3_0_SLS1			    := NOT stSetControl.b3_0_SLS1;
stExpectedStatusData.b3_1_SLS2			    := NOT stSetControl.b3_1_SLS2;
stExpectedStatusData.b3_2_SLS3			    := NOT stSetControl.b3_2_SLS3;
stExpectedStatusData.b3_3_SLS4			    := NOT stSetControl.b3_3_SLS4;
stExpectedStatusData.b3_4_SSR1			    := NOT stSetControl.b3_4_SSR1;
stExpectedStatusData.b3_5_SSR2			    := NOT stSetControl.b3_5_SSR2;
stExpectedStatusData.b3_6_Reserved		    := FALSE;
stExpectedStatusData.b3_7_Reserved		    := FALSE;
stExpectedStatusData.b4_0_SLA1			    := NOT stSetControl.b4_0_SLA1;
stExpectedStatusData.b4_1_SLA2			    := NOT stSetControl.b4_1_SLA2;
stExpectedStatusData.b4_2_SSM1			    := FALSE;
stExpectedStatusData.b4_3_SSM2			    := FALSE;
stExpectedStatusData.b4_4_SSM3			    := FALSE;
stExpectedStatusData.b4_5_SSM4			    := FALSE;
stExpectedStatusData.b4_6_Reserved		    := FALSE;
stExpectedStatusData.b4_7_Reserved		    := FALSE;
stExpectedStatusData.b5_0_Reserved		    := FALSE;
stExpectedStatusData.b5_1_Reserved		    := FALSE;
stExpectedStatusData.b5_2_Reserved		    := FALSE;
stExpectedStatusData.b5_3_Reserved		    := FALSE;
stExpectedStatusData.b5_4_Reserved		    := FALSE;
stExpectedStatusData.b5_5_Reserved		    := FALSE;
stExpectedStatusData.b5_6_Reserved		    := FALSE;
stExpectedStatusData.b5_7_Reserved	        := FALSE;
	
//Act

fbDevice.stControl := stSetControl;
fbDevice.Cycle();
stActualStatusData := fbDevice.stStatus ;

//Assert

AssertEquals(Expected := stExpectedStatusData,
             Actual := stActualStatusData,
             Message := 'Status is not correct');
	 					 			 
TEST_FINISHED();

TEST('Cycle FB Inputs');

//Arrange
stSetControl.b0_0_STO				:=	FALSE;	
stSetControl.b0_1_SLI			    :=  FALSE;
stSetControl.b0_2_SBT			    :=  FALSE;
stSetControl.b0_3_Reserved		    :=  FALSE;
stSetControl.b0_4_MutingEncErr	    :=  FALSE;
stSetControl.b0_5_TestModeActice	:=  FALSE;
stSetControl.b0_6_AckFDI			:=  FALSE;
stSetControl.b0_7_AckError		    :=  FALSE;
stSetControl.b1_0_F_DO0			    :=  FALSE;
stSetControl.b1_1_F_DO1			    :=  FALSE;
stSetControl.b1_2_Reserved		    :=  FALSE;
stSetControl.b1_3_Reserved		    :=  FALSE;
stSetControl.b1_4_Reserved		    :=  FALSE;
stSetControl.b1_5_Reserved		    :=  FALSE;
stSetControl.b1_6_Reserved		    :=  FALSE;
stSetControl.b1_7_Reserved		    :=  FALSE;
stSetControl.b2_0_SOS1			    :=  FALSE;
stSetControl.b2_1_Reserved		    :=  FALSE;
stSetControl.b2_2_SSx1			    :=  FALSE;
stSetControl.b2_3_SSx2			    :=  FALSE;
stSetControl.b2_4_SDI1			    :=  FALSE;
stSetControl.b2_5_SDI2			    :=  FALSE;
stSetControl.b2_6_SLI1			    :=  FALSE;
stSetControl.b2_7_SLI2			    :=  FALSE;
stSetControl.b3_0_SLS1			    :=  FALSE;
stSetControl.b3_1_SLS2			    :=  FALSE;
stSetControl.b3_2_SLS3			    :=  FALSE;
stSetControl.b3_3_SLS4			    :=  FALSE;
stSetControl.b3_4_SSR1			    :=  FALSE;
stSetControl.b3_5_SSR2			    :=  FALSE;
stSetControl.b3_6_Reserved		    :=  FALSE;
stSetControl.b3_7_Reserved		    :=  FALSE;
stSetControl.b4_0_SLA1			    :=  FALSE;
stSetControl.b4_1_SLA2			    :=  FALSE;
stSetControl.b4_2_Reserved		    :=  FALSE;
stSetControl.b4_3_Reserved		    :=  FALSE;
stSetControl.b4_4_Reserved		    :=  FALSE;
stSetControl.b4_5_Reserved		    :=  FALSE;
stSetControl.b4_6_Reserved		    :=  FALSE;
stSetControl.b4_7_Reserved		    :=  FALSE;

fbDevice.bASFDiag := TRUE;
fbDevice.bF_DI0 := TRUE;
fbDevice.bF_DI1 := TRUE;
fbDevice.bF_DI2 := TRUE;
fbDevice.bF_DI3 := TRUE;
fbDevice.bSBTActive := TRUE;
fbDevice.bSSM1 := TRUE;
fbDevice.bSSM2 := TRUE;
fbDevice.bSSM3 := TRUE;
fbDevice.bSSM4 := TRUE;

stExpectedStatusData.b0_0_STOActive			:= stSetControl.b0_0_STO;
stExpectedStatusData.b0_1_ASFDiag		    := TRUE;
stExpectedStatusData.b0_2_SBTActive		    := TRUE;
stExpectedStatusData.b0_3_InputDataValid	:= TRUE;
stExpectedStatusData.b0_4_MutingEncErr	    := stSetControl.b0_4_MutingEncErr;
stExpectedStatusData.b0_5_TestModeActive	:= stSetControl.b0_5_TestModeActice;
stExpectedStatusData.b0_6_Warning		    := FALSE;
stExpectedStatusData.b0_7_ErrorState		:= FALSE;
stExpectedStatusData.b1_0_F_DI0			    := TRUE;
stExpectedStatusData.b1_1_F_DI1			    := TRUE;
stExpectedStatusData.b1_2_F_DI2			    := TRUE;
stExpectedStatusData.b1_3_F_DI3			    := TRUE;
stExpectedStatusData.b1_4_Reserved		    := FALSE;
stExpectedStatusData.b1_5_Reserved		    := FALSE;
stExpectedStatusData.b1_6_Reserved		    := FALSE;
stExpectedStatusData.b1_7_Reserved		    := FALSE;
stExpectedStatusData.b2_0_SOS1			    := NOT stSetControl.b2_0_SOS1;
stExpectedStatusData.b2_1_Reserved		    := FALSE;                  
stExpectedStatusData.b2_2_SSx1			    := NOT stSetControl.b2_2_SSx1;
stExpectedStatusData.b2_3_SSx2			    := NOT stSetControl.b2_3_SSx2;
stExpectedStatusData.b2_4_SDI1			    := NOT stSetControl.b2_4_SDI1;
stExpectedStatusData.b2_5_SDI2			    := NOT stSetControl.b2_5_SDI2;
stExpectedStatusData.b2_6_SLI1			    := NOT stSetControl.b2_6_SLI1;
stExpectedStatusData.b2_7_SLI2			    := NOT stSetControl.b2_7_SLI2;
stExpectedStatusData.b3_0_SLS1			    := NOT stSetControl.b3_0_SLS1;
stExpectedStatusData.b3_1_SLS2			    := NOT stSetControl.b3_1_SLS2;
stExpectedStatusData.b3_2_SLS3			    := NOT stSetControl.b3_2_SLS3;
stExpectedStatusData.b3_3_SLS4			    := NOT stSetControl.b3_3_SLS4;
stExpectedStatusData.b3_4_SSR1			    := NOT stSetControl.b3_4_SSR1;
stExpectedStatusData.b3_5_SSR2			    := NOT stSetControl.b3_5_SSR2;
stExpectedStatusData.b3_6_Reserved		    := FALSE;
stExpectedStatusData.b3_7_Reserved		    := FALSE;
stExpectedStatusData.b4_0_SLA1			    := NOT stSetControl.b4_0_SLA1;
stExpectedStatusData.b4_1_SLA2			    := NOT stSetControl.b4_1_SLA2;
stExpectedStatusData.b4_2_SSM1			    := TRUE;
stExpectedStatusData.b4_3_SSM2			    := TRUE;
stExpectedStatusData.b4_4_SSM3			    := TRUE;
stExpectedStatusData.b4_5_SSM4			    := TRUE;
stExpectedStatusData.b4_6_Reserved		    := FALSE;
stExpectedStatusData.b4_7_Reserved		    := FALSE;
stExpectedStatusData.b5_0_Reserved		    := FALSE;
stExpectedStatusData.b5_1_Reserved		    := FALSE;
stExpectedStatusData.b5_2_Reserved		    := FALSE;
stExpectedStatusData.b5_3_Reserved		    := FALSE;
stExpectedStatusData.b5_4_Reserved		    := FALSE;
stExpectedStatusData.b5_5_Reserved		    := FALSE;
stExpectedStatusData.b5_6_Reserved		    := FALSE;
stExpectedStatusData.b5_7_Reserved	        := FALSE;
	
//Act

fbDevice.stControl := stSetControl;
fbDevice.Cycle();
stActualStatusData := fbDevice.stStatus ;

//Assert

AssertEquals(Expected := stExpectedStatusData,
             Actual := stActualStatusData,
             Message := 'Status is not correct');
	 					 			 
TEST_FINISHED();
END_METHOD

METHOD Test_ProcessDataControl : REFERENCE TO FB_Test
VAR
	fbDevice 					: FB_SEW_Movisafe_CSSx1a;

	stExpectedControlData 		: ST_SEW_Movisafe_CSSx1a_Control;		
	stExpectedControlDataSwap	: ST_SEW_Movisafe_CSSx1a_Control;	
	stActualControlData			: ST_SEW_Movisafe_CSSx1a_Control;	
END_VAR
TEST('Process data to control structure');

//Arrange
stExpectedControlData.b0_0_STO 				:= TRUE;
stExpectedControlData.b0_1_SLI 				:= TRUE;
stExpectedControlData.b0_2_SBT 				:= FALSE;
stExpectedControlData.b0_3_Reserved		    := TRUE;
stExpectedControlData.b0_4_MutingEncErr	    := TRUE;
stExpectedControlData.b0_5_TestModeActice	:= TRUE;
stExpectedControlData.b0_6_AckFDI			:= TRUE;
stExpectedControlData.b0_7_AckError		    := FALSE;
stExpectedControlData.b1_0_F_DO0			:= FALSE;
stExpectedControlData.b1_1_F_DO1			:= TRUE;
stExpectedControlData.b1_2_Reserved		    := TRUE;
stExpectedControlData.b1_3_Reserved		    := FALSE;
stExpectedControlData.b1_4_Reserved		    := TRUE;
stExpectedControlData.b1_5_Reserved		    := TRUE;
stExpectedControlData.b1_6_Reserved		    := FALSE;
stExpectedControlData.b1_7_Reserved		    := TRUE;
stExpectedControlData.b2_0_SOS1			    := TRUE;
stExpectedControlData.b2_1_Reserved		    := FALSE;
stExpectedControlData.b2_2_SSx1			    := FALSE;
stExpectedControlData.b2_3_SSx2			    := FALSE;
stExpectedControlData.b2_4_SDI1			    := TRUE;
stExpectedControlData.b2_5_SDI2			    := TRUE;
stExpectedControlData.b2_6_SLI1			    := TRUE;
stExpectedControlData.b2_7_SLI2			    := FALSE;
stExpectedControlData.b3_0_SLS1			    := TRUE;
stExpectedControlData.b3_1_SLS2			    := TRUE;
stExpectedControlData.b3_2_SLS3			    := TRUE;
stExpectedControlData.b3_3_SLS4			    := TRUE;
stExpectedControlData.b3_4_SSR1			    := TRUE;
stExpectedControlData.b3_5_SSR2			    := TRUE;
stExpectedControlData.b3_6_Reserved		    := TRUE;
stExpectedControlData.b3_7_Reserved		    := FALSE;
stExpectedControlData.b4_0_SLA1			    := FALSE;
stExpectedControlData.b4_1_SLA2			    := TRUE;
stExpectedControlData.b4_2_Reserved		    := TRUE;
stExpectedControlData.b4_3_Reserved		    := TRUE;
stExpectedControlData.b4_4_Reserved		    := TRUE;
stExpectedControlData.b4_5_Reserved		    := FALSE;
stExpectedControlData.b4_6_Reserved		    := TRUE;
stExpectedControlData.b4_7_Reserved		    := FALSE;

fbDevice.pControl := ADR(stExpectedControlData);

//Act
fbDevice.GetControlData();

stActualControlData := fbDevice.stControl;

//Assert
AssertEquals(Expected := stExpectedControlData,
             Actual := stActualControlData,
             Message := 'ControlData is not correct');
	 			 			 
TEST_FINISHED();


TEST('Process data to control structure SWAP');

//Arrange
stExpectedControlData.b0_0_STO 				:= TRUE;
stExpectedControlData.b0_1_SLI 				:= TRUE;
stExpectedControlData.b0_2_SBT 				:= FALSE;
stExpectedControlData.b0_3_Reserved		    := TRUE;
stExpectedControlData.b0_4_MutingEncErr	    := TRUE;
stExpectedControlData.b0_5_TestModeActice	:= TRUE;
stExpectedControlData.b0_6_AckFDI			:= TRUE;
stExpectedControlData.b0_7_AckError		    := FALSE;
stExpectedControlData.b1_0_F_DO0			:= FALSE;
stExpectedControlData.b1_1_F_DO1			:= TRUE;
stExpectedControlData.b1_2_Reserved		    := TRUE;
stExpectedControlData.b1_3_Reserved		    := FALSE;
stExpectedControlData.b1_4_Reserved		    := TRUE;
stExpectedControlData.b1_5_Reserved		    := TRUE;
stExpectedControlData.b1_6_Reserved		    := FALSE;
stExpectedControlData.b1_7_Reserved		    := TRUE;
stExpectedControlData.b2_0_SOS1			    := TRUE;
stExpectedControlData.b2_1_Reserved		    := FALSE;
stExpectedControlData.b2_2_SSx1			    := FALSE;
stExpectedControlData.b2_3_SSx2			    := FALSE;
stExpectedControlData.b2_4_SDI1			    := TRUE;
stExpectedControlData.b2_5_SDI2			    := TRUE;
stExpectedControlData.b2_6_SLI1			    := TRUE;
stExpectedControlData.b2_7_SLI2			    := FALSE;
stExpectedControlData.b3_0_SLS1			    := TRUE;
stExpectedControlData.b3_1_SLS2			    := TRUE;
stExpectedControlData.b3_2_SLS3			    := TRUE;
stExpectedControlData.b3_3_SLS4			    := TRUE;
stExpectedControlData.b3_4_SSR1			    := TRUE;
stExpectedControlData.b3_5_SSR2			    := TRUE;
stExpectedControlData.b3_6_Reserved		    := TRUE;
stExpectedControlData.b3_7_Reserved		    := FALSE;
stExpectedControlData.b4_0_SLA1			    := FALSE;
stExpectedControlData.b4_1_SLA2			    := TRUE;
stExpectedControlData.b4_2_Reserved		    := TRUE;
stExpectedControlData.b4_3_Reserved		    := TRUE;
stExpectedControlData.b4_4_Reserved		    := TRUE;
stExpectedControlData.b4_5_Reserved		    := FALSE;
stExpectedControlData.b4_6_Reserved		    := TRUE;
stExpectedControlData.b4_7_Reserved		    := FALSE;
	
F_Memcpy(ADR(stExpectedControlDataSwap), ADR(stExpectedControlData), SIZEOF(stExpectedControlData), TRUE);

fbDevice.pControl := ADR(stExpectedControlDataSwap);

fbDevice.stConfig.bSwapProcessData := TRUE;

//Act
fbDevice.GetControlData();

stActualControlData := fbDevice.stControl;

//Assert
AssertEquals(Expected := stExpectedControlData,
             Actual := stActualControlData,
             Message := 'CW1 is not correct');

			 			 
TEST_FINISHED();
END_METHOD

METHOD Test_ProcessDataStatus : REFERENCE TO FB_Test
VAR
	fbDevice 						: FB_SEW_Movisafe_CSSx1a;
	
	stExpectedStatusData 			: ST_SEW_Movisafe_CSSx1a_Status;	
	stExpectedStatusDataSwap		: ST_SEW_Movisafe_CSSx1a_Status;
	stActualStatusData 				: ST_SEW_Movisafe_CSSx1a_Status;	
END_VAR
TEST('Assign status structure to process data');

//Arrange
stExpectedStatusData.b0_0_STOActive			:= TRUE;
stExpectedStatusData.b0_1_ASFDiag		    := TRUE;
stExpectedStatusData.b0_2_SBTActive		    := TRUE;
stExpectedStatusData.b0_3_InputDataValid	:= FALSE;
stExpectedStatusData.b0_4_MutingEncErr	    := FALSE;
stExpectedStatusData.b0_5_TestModeActive	:= TRUE;
stExpectedStatusData.b0_6_Warning		    := TRUE;
stExpectedStatusData.b0_7_ErrorState		:= TRUE;
stExpectedStatusData.b1_0_F_DI0			    := FALSE;
stExpectedStatusData.b1_1_F_DI1			    := FALSE;
stExpectedStatusData.b1_2_F_DI2			    := FALSE;
stExpectedStatusData.b1_3_F_DI3			    := TRUE;
stExpectedStatusData.b1_4_Reserved		    := FALSE;
stExpectedStatusData.b1_5_Reserved		    := FALSE;
stExpectedStatusData.b1_6_Reserved		    := TRUE;
stExpectedStatusData.b1_7_Reserved		    := FALSE;
stExpectedStatusData.b2_0_SOS1			    := TRUE;
stExpectedStatusData.b2_1_Reserved		    := TRUE;
stExpectedStatusData.b2_2_SSx1			    := FALSE;
stExpectedStatusData.b2_3_SSx2			    := TRUE;
stExpectedStatusData.b2_4_SDI1			    := TRUE;
stExpectedStatusData.b2_5_SDI2			    := FALSE;
stExpectedStatusData.b2_6_SLI1			    := FALSE;
stExpectedStatusData.b2_7_SLI2			    := FALSE;
stExpectedStatusData.b3_0_SLS1			    := FALSE;
stExpectedStatusData.b3_1_SLS2			    := TRUE;
stExpectedStatusData.b3_2_SLS3			    := FALSE;
stExpectedStatusData.b3_3_SLS4			    := TRUE;
stExpectedStatusData.b3_4_SSR1			    := TRUE;
stExpectedStatusData.b3_5_SSR2			    := TRUE;
stExpectedStatusData.b3_6_Reserved		    := FALSE;
stExpectedStatusData.b3_7_Reserved		    := FALSE;
stExpectedStatusData.b4_0_SLA1			    := TRUE;
stExpectedStatusData.b4_1_SLA2			    := TRUE;
stExpectedStatusData.b4_2_SSM1			    := FALSE;
stExpectedStatusData.b4_3_SSM2			    := TRUE;
stExpectedStatusData.b4_4_SSM3			    := TRUE;
stExpectedStatusData.b4_5_SSM4			    := TRUE;
stExpectedStatusData.b4_6_Reserved		    := TRUE;
stExpectedStatusData.b4_7_Reserved		    := TRUE;
stExpectedStatusData.b5_0_Reserved		    := FALSE;
stExpectedStatusData.b5_1_Reserved		    := TRUE;
stExpectedStatusData.b5_2_Reserved		    := FALSE;
stExpectedStatusData.b5_3_Reserved		    := FALSE;
stExpectedStatusData.b5_4_Reserved		    := FALSE;
stExpectedStatusData.b5_5_Reserved		    := FALSE;
stExpectedStatusData.b5_6_Reserved		    := TRUE;
stExpectedStatusData.b5_7_Reserved		    := FALSE;

fbDevice.pStatus := ADR(stExpectedStatusData);

//Act
fbDevice.SetStatusData();

//Assert
stActualStatusData := fbDevice.stStatus;

AssertEquals(Expected := stExpectedStatusData,
             Actual := stActualStatusData,
             Message := 'Status is not correct');
	 
					 			 
TEST_FINISHED();


TEST('Assign status structure to process data SWAP');

//Arrange
stExpectedStatusData.b0_0_STOActive			:= TRUE;
stExpectedStatusData.b0_1_ASFDiag		    := TRUE;
stExpectedStatusData.b0_2_SBTActive		    := TRUE;
stExpectedStatusData.b0_3_InputDataValid	:= FALSE;
stExpectedStatusData.b0_4_MutingEncErr	    := FALSE;
stExpectedStatusData.b0_5_TestModeActive	:= TRUE;
stExpectedStatusData.b0_6_Warning		    := TRUE;
stExpectedStatusData.b0_7_ErrorState		:= TRUE;
stExpectedStatusData.b1_0_F_DI0			    := FALSE;
stExpectedStatusData.b1_1_F_DI1			    := FALSE;
stExpectedStatusData.b1_2_F_DI2			    := FALSE;
stExpectedStatusData.b1_3_F_DI3			    := TRUE;
stExpectedStatusData.b1_4_Reserved		    := FALSE;
stExpectedStatusData.b1_5_Reserved		    := FALSE;
stExpectedStatusData.b1_6_Reserved		    := TRUE;
stExpectedStatusData.b1_7_Reserved		    := FALSE;
stExpectedStatusData.b2_0_SOS1			    := TRUE;
stExpectedStatusData.b2_1_Reserved		    := TRUE;
stExpectedStatusData.b2_2_SSx1			    := FALSE;
stExpectedStatusData.b2_3_SSx2			    := TRUE;
stExpectedStatusData.b2_4_SDI1			    := TRUE;
stExpectedStatusData.b2_5_SDI2			    := FALSE;
stExpectedStatusData.b2_6_SLI1			    := FALSE;
stExpectedStatusData.b2_7_SLI2			    := FALSE;
stExpectedStatusData.b3_0_SLS1			    := FALSE;
stExpectedStatusData.b3_1_SLS2			    := TRUE;
stExpectedStatusData.b3_2_SLS3			    := FALSE;
stExpectedStatusData.b3_3_SLS4			    := TRUE;
stExpectedStatusData.b3_4_SSR1			    := TRUE;
stExpectedStatusData.b3_5_SSR2			    := TRUE;
stExpectedStatusData.b3_6_Reserved		    := FALSE;
stExpectedStatusData.b3_7_Reserved		    := FALSE;
stExpectedStatusData.b4_0_SLA1			    := TRUE;
stExpectedStatusData.b4_1_SLA2			    := TRUE;
stExpectedStatusData.b4_2_SSM1			    := FALSE;
stExpectedStatusData.b4_3_SSM2			    := TRUE;
stExpectedStatusData.b4_4_SSM3			    := TRUE;
stExpectedStatusData.b4_5_SSM4			    := TRUE;
stExpectedStatusData.b4_6_Reserved		    := TRUE;
stExpectedStatusData.b4_7_Reserved		    := TRUE;
stExpectedStatusData.b5_0_Reserved		    := FALSE;
stExpectedStatusData.b5_1_Reserved		    := TRUE;
stExpectedStatusData.b5_2_Reserved		    := FALSE;
stExpectedStatusData.b5_3_Reserved		    := FALSE;
stExpectedStatusData.b5_4_Reserved		    := FALSE;
stExpectedStatusData.b5_5_Reserved		    := FALSE;
stExpectedStatusData.b5_6_Reserved		    := TRUE;
stExpectedStatusData.b5_7_Reserved		    := FALSE;

F_Memcpy(ADR(stExpectedStatusDataSwap), ADR(stExpectedStatusData), SIZEOF(stExpectedStatusData), TRUE);

fbDevice.pStatus := ADR(stExpectedStatusData);

fbDevice.stConfig.bSwapProcessData := TRUE;

//Act
fbDevice.SetStatusData();

//Assert
stActualStatusData := fbDevice.stStatus;

AssertEquals(Expected := stExpectedStatusData,
             Actual := stActualStatusData,
             Message := 'SW1 is not correct');
	 				 			 
TEST_FINISHED();
END_METHOD

END_FUNCTION_BLOCK

// ---- Devices/SEW_Movisafe_CSSx1a/FB_SEW_Movisafe_CSSx1a.TcPOU
(*
FB_SEW_Movisafe_CSSx1a simulates the funcitionalty of a SEW‑EURODRIVE MOVISAFE® module.

Disclaimer: This simulation is an independent project and is not affiliated with, endorsed by, or approved by SEW‑EURODRIVE. All rights to the SEW‑EURODRIVE brand name and trademarks remain the property of the manufacturer.
Furthermore, no guarantee is given for the completeness of the functional scope or the error-free operation of the simulation. Users should be aware that deviations from the actual product may occur.
*)

{attribute 'reflection'}
FUNCTION_BLOCK FB_SEW_Movisafe_CSSx1a EXTENDS FB_Base IMPLEMENTS I_SEW_Movisafe
VAR_INPUT
	pControl 			: PVOID; //Pocess data from fieldbus. Size must be >= stControl.
	pStatus 			: PVOID; //Pocess data to fieldbus. Size must be >= stStatus.
	stControl 			: ST_SEW_Movisafe_CSSx1a_Control; //Control structure. Is read from the fieldbus.
	stConfig 			: ST_SEW_Movisafe_CSSx1a_Config; //Config structure. Contains parameters of the device.
	
	bASFDiag			: BOOL; //At least one drive safety function has exceeded a limit
	bSBTActive 			: BOOL; //Brake test is active
	bF_DI0				: BOOL; //State digital input 1
	bF_DI1				: BOOL; //State digital input 2
	bF_DI2				: BOOL; //State digital input 3
	bF_DI3				: BOOL; //State digital input 4
	bSSM1				: BOOL; //SSM 1 ist activated (Safe speed monitoring)
	bSSM2				: BOOL; //SSM 2 ist activated (Safe speed monitoring)
	bSSM3				: BOOL;	//SSM 3 ist activated (Safe speed monitoring)
	bSSM4				: BOOL; //SSM 4 ist activated (Safe speed monitoring)
END_VAR

VAR_OUTPUT	
	stStatus			: ST_SEW_Movisafe_CSSx1a_Status;
END_VAR

VAR
    {attribute 'instance-path'} 
    {attribute 'noinit'} 
    _sPath 				: STRING; 
END_VAR

SUPER^();
InitRun();

GetControlData();
Cycle();
SetStatusData();

PROPERTY bSTO : BOOL
GET
bSTO := stStatus.b0_0_StoActive;
END_GET
END_PROPERTY

METHOD Internal Cycle : BOOL
VAR_INPUT
END_VAR
stStatus.b0_0_STOActive			:= stControl.b0_0_STO;
stStatus.b0_1_ASFDiag			:= bASFDiag;
stStatus.b0_2_SBTActive			:= bSBTActive;
stStatus.b0_3_InputDataValid	:= TRUE;
stStatus.b0_4_MutingEncErr		:= stControl.b0_4_MutingEncErr;
stStatus.b0_5_TestModeActive	:= stControl.b0_5_TestModeActice;
stStatus.b0_6_Warning			:= FALSE;
stStatus.b0_7_ErrorState		:= FALSE;
stStatus.b1_0_F_DI0				:= bF_DI0;
stStatus.b1_1_F_DI1				:= bF_DI1;
stStatus.b1_2_F_DI2				:= bF_DI2;
stStatus.b1_3_F_DI3				:= bF_DI3;
stStatus.b1_4_Reserved			:= FALSE;
stStatus.b1_5_Reserved			:= FALSE;
stStatus.b1_6_Reserved			:= FALSE;
stStatus.b1_7_Reserved			:= FALSE;
stStatus.b2_0_SOS1				:= NOT stControl.b2_0_SOS1;
stStatus.b2_1_Reserved			:= FALSE;
stStatus.b2_2_SSx1				:= NOT stControl.b2_2_SSx1;
stStatus.b2_3_SSx2				:= NOT stControl.b2_3_SSx2;
stStatus.b2_4_SDI1				:= NOT stControl.b2_4_SDI1;
stStatus.b2_5_SDI2				:= NOT stControl.b2_5_SDI2;
stStatus.b2_6_SLI1				:= NOT stControl.b2_6_SLI1;
stStatus.b2_7_SLI2				:= NOT stControl.b2_7_SLI2;
stStatus.b3_0_SLS1				:= NOT stControl.b3_0_SLS1;
stStatus.b3_1_SLS2				:= NOT stControl.b3_1_SLS2;
stStatus.b3_2_SLS3				:= NOT stControl.b3_2_SLS3;
stStatus.b3_3_SLS4				:= NOT stControl.b3_3_SLS4;
stStatus.b3_4_SSR1				:= NOT stControl.b3_4_SSR1;
stStatus.b3_5_SSR2				:= NOT stControl.b3_5_SSR2;
stStatus.b3_6_Reserved			:= FALSE;
stStatus.b3_7_Reserved			:= FALSE;
stStatus.b4_0_SLA1				:= NOT stControl.b4_0_SLA1;
stStatus.b4_1_SLA2				:= NOT stControl.b4_1_SLA2;
stStatus.b4_2_SSM1				:= bSSM1;
stStatus.b4_3_SSM2				:= bSSM2;
stStatus.b4_4_SSM3				:= bSSM3;
stStatus.b4_5_SSM4				:= bSSM4;
stStatus.b4_6_Reserved			:= FALSE;
stStatus.b4_7_Reserved			:= FALSE;
stStatus.b5_0_Reserved			:= FALSE;
stStatus.b5_1_Reserved			:= FALSE;
stStatus.b5_2_Reserved			:= FALSE;
stStatus.b5_3_Reserved			:= FALSE;
stStatus.b5_4_Reserved			:= FALSE;
stStatus.b5_5_Reserved			:= FALSE;
stStatus.b5_6_Reserved			:= FALSE;
stStatus.b5_7_Reserved			:= FALSE;
END_METHOD

METHOD INTERNAL GetControlData
VAR_INPUT
END_VAR
IF pControl <= 0 OR stConfig.bForceMode THEN RETURN; END_IF

F_MEMCPY(ADR(stControl), pControl, SIZEOF(stControl), stConfig.bSwapProcessData);
END_METHOD

METHOD INTERNAL InitRun
VAR_INST
	bInitRun : BOOL := TRUE;
END_VAR
IF NOT bInitRun THEN RETURN; END_IF
bInitRun := FALSE;

IF pControl = 0 OR pStatus = 0 THEN
	ADSLOGSTR(ADSLOG_MSGTYPE_WARN, CONCAT(_sPath, ': %s'), 'Plc address not set.');
END_IF
END_METHOD

METHOD INTERNAL SetStatusData
VAR_INPUT
END_VAR
IF pStatus <= 0 THEN RETURN; END_IF

F_MEMCPY(pStatus, ADR(stStatus), SIZEOF(stStatus), stConfig.bSwapProcessData);
END_METHOD

END_FUNCTION_BLOCK

// ---- Tests/Devices/FB_Siemens_RcvDp_Test.TcPOU
FUNCTION_BLOCK FB_Siemens_RcvDp_Test EXTENDS TcUnit.FB_TestSuite

Test_ProcessDataControl();
Test_ProcessDataStatus();

METHOD Test_ProcessDataControl : REFERENCE TO FB_Test
VAR
	fbDevice 						: FB_Siemens_RcvDp;
	
	nExpectdRcvBoolData				: WORD;
	nExpectdRcvInt00				: INT;
	nExpectdRcvInt01				: INT;
	nExpectdRcvData					: WORD;
	nExpectdRcvSequenceNumber		: WORD;
	nExpectdRcvCrc					: WORD;	
	
	nActualRcvBoolData				: WORD;
	nActualRcvInt00					: INT;
	nActualRcvInt01					: INT;
	nActualRcvData					: WORD;
	nActualRcvSequenceNumber		: WORD;
	nActualRcvCrc					: WORD;
		
	stExpectedControlData 			: ST_Siemens_RcvDp_Control;		
	stActualControlData				: ST_Siemens_RcvDp_Control;	
	nDigitalOutputs: INT;
END_VAR
TEST('Process data to control structure');

//Arrange
nExpectdRcvBoolData := 16#A1B2;					
nExpectdRcvInt00 := UINT_TO_INT(16#C3D4);		
nExpectdRcvInt01 := UINT_TO_INT(16#E5F6);		
nExpectdRcvData := 16#B6A5;	
nExpectdRcvSequenceNumber := 16#D4C3;		
nExpectdRcvCrc := 16#E2F1;			

F_Memcpy(ADR(stExpectedControlData), ADR(nExpectdRcvBoolData), 2, FALSE);
F_Memcpy(ADR(stExpectedControlData) + 2, ADR(nExpectdRcvInt00), 2, FALSE);
F_Memcpy(ADR(stExpectedControlData) + 4, ADR(nExpectdRcvInt01), 2, FALSE);
F_Memcpy(ADR(stExpectedControlData) + 6, ADR(nExpectdRcvData), 2, FALSE);
F_Memcpy(ADR(stExpectedControlData) + 8, ADR(nExpectdRcvSequenceNumber), 2, FALSE);
F_Memcpy(ADR(stExpectedControlData) + 10, ADR(nExpectdRcvCrc), 2, FALSE);

fbDevice.pControl := ADR(stExpectedControlData);

//Act
fbDevice.GetControlData();

stActualControlData := fbDevice.stControl;

//Assert

AssertEquals(Expected := nExpectdRcvBoolData,
             Actual := stActualControlData.nRcvBoolData,
             Message := 'RcvBoolData is not correct');
	 
AssertEquals(Expected := nExpectdRcvInt00,
             Actual := stActualControlData.nRcvInt00,
             Message := 'RcvInt00 is not correct');
			 
AssertEquals(Expected := nExpectdRcvInt01,
             Actual := stActualControlData.nRcvInt01,
             Message := 'RcvInt01 is not correct');
			 
AssertEquals(Expected := nExpectdRcvData,
             Actual := stActualControlData.nRcvData,
             Message := 'RcvData is not correct');
			 
AssertEquals(Expected := nExpectdRcvSequenceNumber,
             Actual := stActualControlData.nRcvSequenceNumber,
             Message := 'SequenceNumber is not correct');
			 
AssertEquals(Expected := nExpectdRcvCrc,
             Actual := stActualControlData.nRcvCrc,
             Message := 'RcvCrc is not correct');			 
			 
TEST_FINISHED();


TEST('Process data to control structure SWAP');
//Arrange
nExpectdRcvBoolData := 16#A1B2;					
nExpectdRcvInt00 := UINT_TO_INT(16#C3D4);		
nExpectdRcvInt01 := UINT_TO_INT(16#E5F6);		
nExpectdRcvData := 16#B6A5;	
nExpectdRcvSequenceNumber := 16#D4C3;		
nExpectdRcvCrc := 16#E2F1;			

F_Memcpy(ADR(stExpectedControlData), ADR(nExpectdRcvBoolData), 2, TRUE);
F_Memcpy(ADR(stExpectedControlData) + 2, ADR(nExpectdRcvInt00), 2, TRUE);
F_Memcpy(ADR(stExpectedControlData) + 4, ADR(nExpectdRcvInt01), 2, TRUE);
F_Memcpy(ADR(stExpectedControlData) + 6, ADR(nExpectdRcvData), 2, TRUE);
F_Memcpy(ADR(stExpectedControlData) + 8, ADR(nExpectdRcvSequenceNumber), 2, TRUE);
F_Memcpy(ADR(stExpectedControlData) + 10, ADR(nExpectdRcvCrc), 2, TRUE);

fbDevice.pControl := ADR(stExpectedControlData);

fbDevice.stConfig.bSwapProcessData := TRUE;

//Act
fbDevice.GetControlData();

stActualControlData := fbDevice.stControl;

//Assert

AssertEquals(Expected := nExpectdRcvBoolData,
             Actual := stActualControlData.nRcvBoolData,
             Message := 'RcvBoolData is not correct');
	 
AssertEquals(Expected := nExpectdRcvInt00,
             Actual := stActualControlData.nRcvInt00,
             Message := 'RcvInt00 is not correct');
			 
AssertEquals(Expected := nExpectdRcvInt01,
             Actual := stActualControlData.nRcvInt01,
             Message := 'RcvInt01 is not correct');
			 
AssertEquals(Expected := nExpectdRcvData,
             Actual := stActualControlData.nRcvData,
             Message := 'RcvData is not correct');
			 
AssertEquals(Expected := nExpectdRcvSequenceNumber,
             Actual := stActualControlData.nRcvSequenceNumber,
             Message := 'SequenceNumber is not correct');
			 
AssertEquals(Expected := nExpectdRcvCrc,
             Actual := stActualControlData.nRcvCrc,
             Message := 'RcvCrc is not correct');			 
			 
TEST_FINISHED();
END_METHOD

METHOD Test_ProcessDataStatus : REFERENCE TO FB_Test
VAR
	fbDevice 						: FB_Siemens_RcvDp;
	
	nExpectedSendData				: WORD;
	nExpectedSendSequenceNumber		: WORD;	
	nExpectedSendCrc				: WORD;
	
	//nActualSendData					: WORD;
	//nActualSendSequenceNumber		: WORD;	
	//nActualSendCrc					: WORD;

	stExpectedStatusData 			: ST_Siemens_RcvDp_Status;		
	stActualStatusData 				: ST_Siemens_RcvDp_Status;	
END_VAR
TEST('Assign status structure to process data');

//Arrange
nExpectedSendData := 16#A1B2;					
nExpectedSendSequenceNumber := 16#C3D4;		
nExpectedSendCrc := 16#E5F6;		
		
	
F_Memcpy(ADR(fbDevice.stStatus), ADR(nExpectedSendData), 2, FALSE);
F_Memcpy(ADR(fbDevice.stStatus) + 2, ADR(nExpectedSendSequenceNumber), 2, FALSE);
F_Memcpy(ADR(fbDevice.stStatus) + 4, ADR(nExpectedSendCrc), 2, FALSE);

fbDevice.pStatus := ADR(stActualStatusData);

//Act
fbDevice.SetStatusData();

//Assert
//F_Memcpy(ADR(nActualSendData), ADR(stActualStatusData), 2, FALSE);
//F_Memcpy(ADR(nActualSendSequenceNumber), ADR(stActualStatusData) + 2, 2, FALSE);
//F_Memcpy(ADR(nActualSendCrc), ADR(stActualStatusData) + 4, 2, FALSE);

AssertEquals(Expected := nExpectedSendData,
             Actual := stActualStatusData.nSendData,
             Message := 'SendData is not correct');
	 
AssertEquals(Expected := nExpectedSendSequenceNumber,
             Actual := stActualStatusData.nSendSequenceNumber,
             Message := 'SendSequenceNumber is not correct');	

AssertEquals(Expected := nExpectedSendCrc,
             Actual := stActualStatusData.nSendCrc,
             Message := 'SendCrc is not correct');
					 			 
TEST_FINISHED();


TEST('Assign status structure to process data SWAP');

//Arrange
nExpectedSendData := 16#A1B2;					
nExpectedSendSequenceNumber := 16#C3D4;		
nExpectedSendCrc := 16#E5F6;		
		
F_Memcpy(ADR(fbDevice.stStatus), ADR(nExpectedSendData), 2, TRUE);
F_Memcpy(ADR(fbDevice.stStatus) + 2, ADR(nExpectedSendSequenceNumber), 2, TRUE);
F_Memcpy(ADR(fbDevice.stStatus) + 4, ADR(nExpectedSendCrc), 2, TRUE);

fbDevice.pStatus := ADR(stActualStatusData);

fbDevice.stConfig.bSwapProcessData := TRUE;

//Act
fbDevice.SetStatusData();

//Assert
//F_Memcpy(ADR(nActualSendData), ADR(stActualStatusData), 2, FALSE);
//F_Memcpy(ADR(nActualSendSequenceNumber), ADR(stActualStatusData) + 2, 2, FALSE);
//F_Memcpy(ADR(nActualSendCrc), ADR(stActualStatusData) + 4, 2, FALSE);

AssertEquals(Expected := nExpectedSendData,
             Actual := stActualStatusData.nSendData,
             Message := 'SendData is not correct');
	 
AssertEquals(Expected := nExpectedSendSequenceNumber,
             Actual := stActualStatusData.nSendSequenceNumber,
             Message := 'SendSequenceNumber is not correct');	

AssertEquals(Expected := nExpectedSendCrc,
             Actual := stActualStatusData.nSendCrc,
             Message := 'SendCrc is not correct');
TEST_FINISHED();
END_METHOD

END_FUNCTION_BLOCK

// ---- Devices/Siemens_RcvDp/FB_Siemens_RcvDp.TcPOU
(*
FB_Siemens_RcvDp simulates the funcitionalty of a Siemens PN/PN coupler RCVDP safety-related communication.

Disclaimer: This simulation is an independent project and is not affiliated with, endorsed by, or approved by Siemens. All rights to the Siemens brand name and trademarks remain the property of the manufacturer.
Furthermore, no guarantee is given for the completeness of the functional scope or the error-free operation of the simulation. Users should be aware that deviations from the actual product may occur.
*)

{attribute 'reflection'} 
FUNCTION_BLOCK FB_Siemens_RcvDp EXTENDS FB_Base
VAR_INPUT
	pControl 			: PVOID; //Pocess data from fieldbus. Size must be >= stControl.
	pStatus 			: PVOID; //Pocess data to fieldbus. Size must be >= stStatus.
	stControl			: ST_Siemens_RcvDp_Control; 
	stConfig 			: ST_Siemens_RcvDp_Config;
	
	stDevData			: ST_Siemens_RcvDp_DevData;
END_VAR

VAR_OUTPUT
	stStatus			: ST_Siemens_RcvDp_Status; 
	
	stHstData			: ST_Siemens_RcvDp_HstData;
END_VAR

VAR
    {attribute 'instance-path'} 
    {attribute 'noinit'} 
    _sPath 				: STRING; 

	_nLastSequenceNumber: WORD;
	_nCalculatedCrc		: WORD;	
	_TonTimeout			: TON;	
END_VAR

VAR CONSTANT
	N_POLYNOM			: WORD := 16#4EAB;
END_VAR

SUPER^();
InitRun();	
GetControlData();
Cycle();
SetStatusData();

METHOD PRIVATE Cycle
VAR_INPUT
END_VAR
(* Simplified communication when using PLCSIM Adv. *)
	IF OC_Core.GVL_Core.fbSystem.eControllerType = E_ControllerType.PlcSimAdvanced THEN
		SimLogic();
		RETURN;
	END_IF

(* Calculate received crc *)
	_nCalculatedCrc := F_CalcCrc16(ADR(stControl), 8, stConfig.nDpDpId, N_POLYNOM);

(* Restart timer, if sequence number has changed *)
	IF stControl.nRcvSequenceNumber <> _nLastSequenceNumber AND NOT stHstData.bError THEN
		_nLastSequenceNumber := stControl.nRcvSequenceNumber;
		stHstData.bSubsOn	:= FALSE;
		_TonTimeout.IN		:= FALSE;
	ELSE
		_TonTimeout.IN		:= TRUE;
	END_IF

(* Reintegration *)
	IF (stConfig.bAutoAckRei AND stHstData.bError) OR stDevData.bAckRei THEN
		stHstData.bError 	:= FALSE;
		_TonTimeout.IN		:= FALSE;
	END_IF

(* Check if timer has expired *)
	_TonTimeout();
	
	IF _TonTimeout.Q	THEN
		stHstData.bError	:= TRUE;
		stHstData.bSubsOn	:= TRUE;
	END_IF

(* compare received crc value with calculated crc *)
	IF stControl.nRcvCrc = _nCalculatedCrc AND NOT stHstData.bError THEN
		stHstData.bSubsOn	:= FALSE;
	ELSE
		stHstData.bError	:= TRUE;
		stHstData.bSubsOn	:= TRUE;
	END_IF

(* Get substitude or safety values *)
	IF stHstData.bSubsOn THEN
		stHstData.bRcv00	:= stDevData.bSub00;
		stHstData.bRcv01	:= stDevData.bSub01;
		stHstData.bRcv02	:= stDevData.bSub02;
		stHstData.bRcv03	:= stDevData.bSub03;
		stHstData.bRcv04	:= stDevData.bSub04;
		stHstData.bRcv05	:= stDevData.bSub05;
		stHstData.bRcv06	:= stDevData.bSub06;
		stHstData.bRcv07	:= stDevData.bSub07;
		stHstData.bRcv08	:= stDevData.bSub08;
		stHstData.bRcv09	:= stDevData.bSub09;
		stHstData.bRcv10	:= stDevData.bSub10;
		stHstData.bRcv11	:= stDevData.bSub11;
		stHstData.bRcv12	:= stDevData.bSub12;
		stHstData.bRcv13	:= stDevData.bSub13;
		stHstData.bRcv14	:= stDevData.bSub14;
		stHstData.bRcv15	:= stDevData.bSub15;
		stHstData.nRcv00	:= stDevData.nSub00;
		stHstData.nRcv01	:= stDevData.nSub01;
	ELSE
		stHstData.bRcv00	:= stControl.nRcvBoolData.0;
		stHstData.bRcv01	:= stControl.nRcvBoolData.1;
		stHstData.bRcv02	:= stControl.nRcvBoolData.2;
		stHstData.bRcv03	:= stControl.nRcvBoolData.3;
		stHstData.bRcv04	:= stControl.nRcvBoolData.4;
		stHstData.bRcv05	:= stControl.nRcvBoolData.5;
		stHstData.bRcv06	:= stControl.nRcvBoolData.6;
		stHstData.bRcv07	:= stControl.nRcvBoolData.7;
		stHstData.bRcv08	:= stControl.nRcvBoolData.8;  
		stHstData.bRcv09	:= stControl.nRcvBoolData.9;  
		stHstData.bRcv10	:= stControl.nRcvBoolData.10;  
		stHstData.bRcv11	:= stControl.nRcvBoolData.11;  
		stHstData.bRcv12	:= stControl.nRcvBoolData.12; 
		stHstData.bRcv13	:= stControl.nRcvBoolData.13; 
		stHstData.bRcv14	:= stControl.nRcvBoolData.14; 
		stHstData.bRcv15	:= stControl.nRcvBoolData.15;	
		stHstData.nRcv00	:= stControl.nRcvInt00;
		stHstData.nRcv01	:= stControl.nRcvInt01;
	END_IF

(* Send data *)
	stStatus.nSendData				:= BOOL_TO_WORD(stHstData.bSubsOn);
	stStatus.nSendSequenceNumber	:= stControl.nRcvSequenceNumber;
	stStatus.nSendCrc 				:= F_CalcCrc16(ADR(stStatus.nSendData), 2, stConfig.nDpDpId, N_POLYNOM);
END_METHOD

METHOD INTERNAL GetControlData
VAR_INPUT
END_VAR
IF pControl <= 0 OR stConfig.bForceMode THEN RETURN; END_IF

// nRcvBoolData
F_Memcpy(ADR(stControl), pControl, 2, stConfig.bSwapProcessData);
// nRcvInt00
F_Memcpy(ADR(stControl) + 2, pControl + 2, 2, stConfig.bSwapProcessData);		
// nRcvInt01
F_Memcpy(ADR(stControl) + 4, pControl + 4, 2, stConfig.bSwapProcessData);			
// nRcvData
F_Memcpy(ADR(stControl) + 6, pControl + 6, 2, stConfig.bSwapProcessData);			
// nRcvSequenceNumber
F_Memcpy(ADR(stControl) + 8, pControl + 8, 2, stConfig.bSwapProcessData);	
// nRcvCrc
F_Memcpy(ADR(stControl) + 10, pControl + 10, 2, stConfig.bSwapProcessData);
END_METHOD

METHOD INTERNAL InitRun : BOOL
VAR_INST
	bInitRun : BOOL := TRUE;
END_VAR
IF NOT bInitRun THEN RETURN; END_IF
bInitRun := FALSE;

IF pControl = 0 OR pStatus = 0 THEN
	ADSLOGSTR(ADSLOG_MSGTYPE_WARN, CONCAT(_sPath, ': %s'), 'Plc address not set.');
END_IF

_TonTimeout.PT := REAL_TO_TIME(stConfig.fTimeout);
END_METHOD

METHOD INTERNAL SetStatusData
VAR_INPUT
END_VAR
IF pStatus <= 0 THEN RETURN; END_IF


// nSendData
F_Memcpy(pStatus, ADR(stStatus), 2, stConfig.bSwapProcessData);				
// nSendSequenceNumber
F_Memcpy(pStatus + 2, ADR(stStatus) + 2, 2, stConfig.bSwapProcessData);
// nSendCrc
F_Memcpy(pStatus + 4, ADR(stStatus) + 4, 2, stConfig.bSwapProcessData);
END_METHOD

METHOD PRIVATE SimLogic
VAR_INPUT
END_VAR
(* No error or substitude values in sim mode *)
	stHstData.bError 	:= FALSE;
	stHstData.bSubsOn	:= FALSE;

(* Get safety values *)
	stHstData.bRcv00	:= stControl.nRcvBoolData.0;
	stHstData.bRcv01	:= stControl.nRcvBoolData.1;
	stHstData.bRcv02	:= stControl.nRcvBoolData.2;
	stHstData.bRcv03	:= stControl.nRcvBoolData.3;
	stHstData.bRcv04	:= stControl.nRcvBoolData.4;
	stHstData.bRcv05	:= stControl.nRcvBoolData.5;
	stHstData.bRcv06	:= stControl.nRcvBoolData.6;
	stHstData.bRcv07	:= stControl.nRcvBoolData.7;
	stHstData.bRcv08	:= stControl.nRcvBoolData.8;  
	stHstData.bRcv09	:= stControl.nRcvBoolData.9;  
	stHstData.bRcv10	:= stControl.nRcvBoolData.10;  
	stHstData.bRcv11	:= stControl.nRcvBoolData.11;  
	stHstData.bRcv12	:= stControl.nRcvBoolData.12; 
	stHstData.bRcv13	:= stControl.nRcvBoolData.13; 
	stHstData.bRcv14	:= stControl.nRcvBoolData.14; 
	stHstData.bRcv15	:= stControl.nRcvBoolData.15;	
	stHstData.nRcv00	:= stControl.nRcvInt00;
	stHstData.nRcv01	:= stControl.nRcvInt01;

(* Send data *)
	stStatus.nSendData				:= 16#80;
	stStatus.nSendSequenceNumber	:= stControl.nRcvSequenceNumber;
	stStatus.nSendCrc 				:= F_CalcCrc16(ADR(stStatus.nSendData), 2, stConfig.nDpDpId, N_POLYNOM);
END_METHOD

END_FUNCTION_BLOCK

// ---- Common/Utils/F_CalcCrc16.TcPOU
FUNCTION F_CalcCrc16 : WORD
VAR_INPUT
	pData		: POINTER TO BYTE;
	nDataSize	: INT;
	nInitCRC	: WORD;
	nPolynom	: WORD;
END_VAR
VAR
	nCrc		: WORD;
	nDataX		: BYTE;
	nI			: INT;
	nJ			: INT;
END_VAR

nCrc := nInitCRC;

FOR nI := 0 TO nDataSize - 1 BY 1 DO
	nDataX	:= pData[nI];
	FOR nJ := 0 TO 7 BY 1 DO
		IF (SHR(nCrc,15) AND 1) <> (SHR(nDataX,7) AND 1) THEN
			nCrc := SHL(nCrc,1) XOR nPolynom;
		ELSE
			nCrc := SHL(nCrc,1);
		END_IF
		nDataX := SHL(nDataX,1);
	END_FOR	
END_FOR

F_CalcCrc16 := nCrc;

END_FUNCTION

// ---- Tests/Devices/FB_Siemens_SendDp_Test.TcPOU
FUNCTION_BLOCK FB_Siemens_SendDp_Test EXTENDS TcUnit.FB_TestSuite

Test_ProcessDataControl();
Test_ProcessDataStatus();

METHOD Test_ProcessDataControl : REFERENCE TO FB_Test
VAR
	fbDevice 						: FB_Siemens_SendDp;
	
	nExpectdRcvData					: WORD;
	nExpectdRcvSequenceNumber		: WORD;
	nExpectdRcvCrc					: WORD;	
	
	nActualRcvData					: WORD;
	nActualRcvSequenceNumber		: WORD;
	nActualRcvCrc					: WORD;
		
	stExpectedControlData 			: ST_Siemens_SendDp_Control;		
	stActualControlData				: ST_Siemens_SendDp_Control;	
	nDigitalOutputs: INT;
END_VAR
TEST('Process data to control structure');

//Arrange
nExpectdRcvData := 16#A1B2;					
nExpectdRcvSequenceNumber := 16#C3D4;		
nExpectdRcvCrc := 16#E5F6;		
	
F_Memcpy(ADR(stExpectedControlData), ADR(nExpectdRcvData), 2, FALSE);
F_Memcpy(ADR(stExpectedControlData) + 2, ADR(nExpectdRcvSequenceNumber), 2, FALSE);
F_Memcpy(ADR(stExpectedControlData) + 4, ADR(nExpectdRcvCrc), 2, FALSE);

fbDevice.pControl := ADR(stExpectedControlData);

//Act
fbDevice.GetControlData();

stActualControlData := fbDevice.stControl;

//Assert
			 
AssertEquals(Expected := nExpectdRcvData,
             Actual := stActualControlData.nRcvData,
             Message := 'RcvData is not correct');
			 
AssertEquals(Expected := nExpectdRcvSequenceNumber,
             Actual := stActualControlData.nRcvSequenceNumber,
             Message := 'SequenceNumber is not correct');
			 
AssertEquals(Expected := nExpectdRcvCrc,
             Actual := stActualControlData.nRcvCrc,
             Message := 'RcvCrc is not correct');			 
			 
TEST_FINISHED();


TEST('Process data to control structure SWAP');

//Arrange
nExpectdRcvData := 16#A1B2;					
nExpectdRcvSequenceNumber := 16#C3D4;		
nExpectdRcvCrc := 16#E5F6;		
	
F_Memcpy(ADR(stExpectedControlData), ADR(nExpectdRcvData), 2, TRUE);
F_Memcpy(ADR(stExpectedControlData) + 2, ADR(nExpectdRcvSequenceNumber), 2, TRUE);
F_Memcpy(ADR(stExpectedControlData) + 4, ADR(nExpectdRcvCrc), 2, TRUE);

fbDevice.pControl := ADR(stExpectedControlData);

fbDevice.stConfig.bSwapProcessData := TRUE;

//Act
fbDevice.GetControlData();

stActualControlData := fbDevice.stControl;

//Assert
			 
AssertEquals(Expected := nExpectdRcvData,
             Actual := stActualControlData.nRcvData,
             Message := 'RcvData is not correct');
			 
AssertEquals(Expected := nExpectdRcvSequenceNumber,
             Actual := stActualControlData.nRcvSequenceNumber,
             Message := 'SequenceNumber is not correct');
			 
AssertEquals(Expected := nExpectdRcvCrc,
             Actual := stActualControlData.nRcvCrc,
             Message := 'RcvCrc is not correct');				 
			 
TEST_FINISHED();
END_METHOD

METHOD Test_ProcessDataStatus : REFERENCE TO FB_Test
VAR
	fbDevice 						: FB_Siemens_SendDp;
	
	nExpectedBoolData				: WORD;
	nExpectedSendInt00				: INT;
	nExpectedSendInt01				: INT;
	nExpectedSendData				: WORD;
	nExpectedSendSequenceNumber		: WORD;	
	nExpectedSendCrc				: WORD;
	
	stExpectedStatusData 			: ST_Siemens_SendDp_Status;		
	stActualStatusData 				: ST_Siemens_SendDp_Status;	
END_VAR
TEST('Assign status structure to process data');

//Arrange
nExpectedBoolData := 16#A1B2;	
nExpectedSendInt00 := UINT_TO_INT(16#C3D4);
nExpectedSendInt01 := UINT_TO_INT(16#E5F6);	
nExpectedSendData := 16#B6A5;					
nExpectedSendSequenceNumber := 16#D4C3;	
nExpectedSendCrc := 16#E2F1;		

F_Memcpy(ADR(fbDevice.stStatus), ADR(nExpectedBoolData), 2, FALSE);
F_Memcpy(ADR(fbDevice.stStatus) + 2, ADR(nExpectedSendInt00), 2, FALSE);
F_Memcpy(ADR(fbDevice.stStatus) + 4, ADR(nExpectedSendInt01), 2, FALSE);
F_Memcpy(ADR(fbDevice.stStatus) + 6, ADR(nExpectedSendData), 2, FALSE);
F_Memcpy(ADR(fbDevice.stStatus) + 8, ADR(nExpectedSendSequenceNumber), 2, FALSE);
F_Memcpy(ADR(fbDevice.stStatus) + 10, ADR(nExpectedSendCrc), 2, FALSE);

fbDevice.pStatus := ADR(stActualStatusData);

//Act
fbDevice.SetStatusData();

//Assert
AssertEquals(Expected := nExpectedBoolData,
             Actual := stActualStatusData.nSendBoolData,
             Message := 'SendBoolData is not correct');
	 
AssertEquals(Expected := nExpectedSendInt00,
             Actual := stActualStatusData.nSendInt00,
             Message := 'SendInt00 is not correct');	

AssertEquals(Expected := nExpectedSendInt01,
             Actual := stActualStatusData.nSendInt01,
             Message := 'SendInt01 is not correct');
			 
AssertEquals(Expected := nExpectedSendData,
             Actual := stActualStatusData.nSendData,
             Message := 'SendData is not correct');
	 
AssertEquals(Expected := nExpectedSendSequenceNumber,
             Actual := stActualStatusData.nSendSequenceNumber,
             Message := 'SendSequenceNumber is not correct');	

AssertEquals(Expected := nExpectedSendCrc,
             Actual := stActualStatusData.nSendCrc,
             Message := 'SendCrc is not correct');
					 			 
TEST_FINISHED();


TEST('Assign status structure to process data SWAP');

//Arrange
nExpectedBoolData := 16#A1B2;	
nExpectedSendInt00 := UINT_TO_INT(16#C3D4);
nExpectedSendInt01 := UINT_TO_INT(16#E5F6);	
nExpectedSendData := 16#B6A5;					
nExpectedSendSequenceNumber := 16#D4C3;	
nExpectedSendCrc := 16#E2F1;		

F_Memcpy(ADR(fbDevice.stStatus), ADR(nExpectedBoolData), 2, TRUE);
F_Memcpy(ADR(fbDevice.stStatus) + 2, ADR(nExpectedSendInt00), 2, TRUE);
F_Memcpy(ADR(fbDevice.stStatus) + 4, ADR(nExpectedSendInt01), 2, TRUE);
F_Memcpy(ADR(fbDevice.stStatus) + 6, ADR(nExpectedSendData), 2, TRUE);
F_Memcpy(ADR(fbDevice.stStatus) + 8, ADR(nExpectedSendSequenceNumber), 2, TRUE);
F_Memcpy(ADR(fbDevice.stStatus) + 10, ADR(nExpectedSendCrc), 2, TRUE);

fbDevice.pStatus := ADR(stActualStatusData);

fbDevice.stConfig.bSwapProcessData := TRUE;

//Act
fbDevice.SetStatusData();

//Assert
AssertEquals(Expected := nExpectedBoolData,
             Actual := stActualStatusData.nSendBoolData,
             Message := 'SendBoolData is not correct');
	 
AssertEquals(Expected := nExpectedSendInt00,
             Actual := stActualStatusData.nSendInt00,
             Message := 'SendInt00 is not correct');	

AssertEquals(Expected := nExpectedSendInt01,
             Actual := stActualStatusData.nSendInt01,
             Message := 'SendInt01 is not correct');
			 
AssertEquals(Expected := nExpectedSendData,
             Actual := stActualStatusData.nSendData,
             Message := 'SendData is not correct');
	 
AssertEquals(Expected := nExpectedSendSequenceNumber,
             Actual := stActualStatusData.nSendSequenceNumber,
             Message := 'SendSequenceNumber is not correct');	

AssertEquals(Expected := nExpectedSendCrc,
             Actual := stActualStatusData.nSendCrc,
             Message := 'SendCrc is not correct');
					 			 
TEST_FINISHED();
END_METHOD

END_FUNCTION_BLOCK

// ---- Devices/Siemens_SendDp/FB_Siemens_SendDp.TcPOU
(*
FB_Siemens_SendDp simulates the funcitionalty of a Siemens PN/PN coupler SENDDP safety-related communication.

Disclaimer: This simulation is an independent project and is not affiliated with, endorsed by, or approved by Siemens. All rights to the Siemens brand name and trademarks remain the property of the manufacturer.
Furthermore, no guarantee is given for the completeness of the functional scope or the error-free operation of the simulation. Users should be aware that deviations from the actual product may occur.
*)

{attribute 'reflection'} 
FUNCTION_BLOCK FB_Siemens_SendDp EXTENDS FB_Base
VAR_INPUT
	pControl 			: PVOID; //Pocess data from fieldbus. Size must be >= stControl.
	pStatus 			: PVOID; //Pocess data to fieldbus. Size must be >= stStatus.
	stControl				: ST_Siemens_SendDp_Control; 	
	stConfig 			: ST_Siemens_SendDp_Config;
	
	stDevData			: ST_Siemens_SendDp_DevData;
END_VAR

VAR_OUTPUT
	stStatus			: ST_Siemens_SendDp_Status; 	

	stHstData			: ST_Siemens_SendDp_HstData;
END_VAR

VAR
    {attribute 'instance-path'} 
    {attribute 'noinit'} 
    _sPath 				: STRING; 
	
	_nLastSequenceNumber	: WORD;
	_nSendSequenceNumber	: WORD;
	_nCalculatedCrc		: WORD;	
	_TonTimeout			: TON;
END_VAR

VAR CONSTANT
	POLYNOM			: WORD := 16#4EAB;
END_VAR

SUPER^();
InitRun();
GetControlData();
Cycle();
SetStatusData();

METHOD PRIVATE Cycle
(* Simplified communication when using PLCSIM Adv. *)
	IF OC_Core.GVL_Core.fbSystem.eControllerType = E_ControllerType.PlcSimAdvanced THEN
		SimLogic();
		RETURN;
	END_IF

(* Calculate received crc *)
	_nCalculatedCrc := F_CalcCrc16(ADR(stControl), 2, stConfig.nDpDpId, POLYNOM);

(* Restart timer, if sequence number has changed *)
	IF stControl.nRcvSequenceNumber <> _nLastSequenceNumber THEN
		_TonTimeout.IN		:= FALSE;
		_nLastSequenceNumber := stControl.nRcvSequenceNumber;
		stHstData.bError	:= FALSE;
		stHstData.bSubsOn	:= FALSE;
	ELSE
		_TonTimeout.IN		:= TRUE;
	END_IF

(* Check if timer has expired *)
	_TonTimeout();
	
	IF _TonTimeout.Q	THEN
		_TonTimeout.IN		:= FALSE;
		_nSendSequenceNumber := 0;
		stHstData.bError	:= TRUE;
		stHstData.bSubsOn	:= TRUE;
	END_IF

(* compare received crc value with calculated crc *)
	IF stControl.nRcvCrc = _nCalculatedCrc THEN
		IF _nSendSequenceNumber = stControl.nRcvSequenceNumber THEN
			IF _nSendSequenceNumber = 0 THEN
				_nSendSequenceNumber := 1;
			ELSE
				_nSendSequenceNumber := _nSendSequenceNumber + 1;
			END_IF
		END_IF
	END_IF

(* Limit sequence number to 32767 *)
	IF _nSendSequenceNumber > 32767 THEN
		_nSendSequenceNumber := 1;
	END_IF

(* Send data *)
	stStatus.nSendBoolData.0 		:= stDevData.bSend00;
	stStatus.nSendBoolData.1 		:= stDevData.bSend01;
	stStatus.nSendBoolData.2 		:= stDevData.bSend02;
	stStatus.nSendBoolData.3 		:= stDevData.bSend03;
	stStatus.nSendBoolData.4 		:= stDevData.bSend04;
	stStatus.nSendBoolData.5 		:= stDevData.bSend05;
	stStatus.nSendBoolData.6 		:= stDevData.bSend06;
	stStatus.nSendBoolData.7 		:= stDevData.bSend07;
	stStatus.nSendBoolData.8 		:= stDevData.bSend08;
	stStatus.nSendBoolData.9 		:= stDevData.bSend09;
	stStatus.nSendBoolData.10 		:= stDevData.bSend10;
	stStatus.nSendBoolData.11 		:= stDevData.bSend11;
	stStatus.nSendBoolData.12 		:= stDevData.bSend12;
	stStatus.nSendBoolData.13 		:= stDevData.bSend13;
	stStatus.nSendBoolData.14 		:= stDevData.bSend14;
	stStatus.nSendBoolData.15 		:= stDevData.bSend15;
	stStatus.nSendInt00				:= stDevData.nSend00;
	stStatus.nSendInt01				:= stDevData.nSend01;
	stStatus.nSendData				:= BOOL_TO_WORD(stHstData.bSubsOn);
	stStatus.nSendSequenceNumber 	:= _nSendSequenceNumber;
	stStatus.nSendCrc 				:= F_CalcCrc16(ADR(stStatus), 8, stConfig.nDpDpId, POLYNOM);
END_METHOD

METHOD INTERNAL GetControlData
VAR_INPUT
END_VAR
IF pControl <= 0 OR stConfig.bForceMode THEN RETURN; END_IF

// nRcvData
F_Memcpy(ADR(stControl), pControl, 2, stConfig.bSwapProcessData);
// nRcvSequenceNumber
F_Memcpy(ADR(stControl) + 2, pControl + 2, 2, stConfig.bSwapProcessData);
// nRcvCrc
F_Memcpy(ADR(stControl) + 4, pControl + 4, 2, stConfig.bSwapProcessData);
END_METHOD

METHOD INTERNAL InitRun : BOOL
VAR_INST
	bInitRun : BOOL := TRUE;
END_VAR
IF NOT bInitRun THEN RETURN; END_IF
bInitRun := FALSE;

IF pControl = 0 OR pStatus = 0 THEN
	ADSLOGSTR(ADSLOG_MSGTYPE_WARN, CONCAT(_sPath, ': %s'), 'Plc address not set.');
END_IF

_TonTimeout.PT := REAL_TO_TIME(stConfig.fTimeout);
END_METHOD

METHOD INTERNAL SetStatusData
VAR_INPUT
END_VAR
IF pStatus <= 0 THEN RETURN; END_IF

// nSendBoolData
F_Memcpy(pStatus, ADR(stStatus), 2, stConfig.bSwapProcessData);
// nSendInt00
F_Memcpy(pStatus + 2, ADR(stStatus) + 2, 2, stConfig.bSwapProcessData);		
// nSendInt01
F_Memcpy(pStatus + 4, ADR(stStatus) + 4, 2, stConfig.bSwapProcessData);		
// nSendData
F_Memcpy(pStatus + 6, ADR(stStatus) + 6, 2, stConfig.bSwapProcessData);	
// nSendSequenceNumber
F_Memcpy(pStatus + 8, ADR(stStatus) + 8, 2, stConfig.bSwapProcessData);
// nSendCrc
F_Memcpy(pStatus + 10, ADR(stStatus) + 10, 2, stConfig.bSwapProcessData);
END_METHOD

METHOD PRIVATE SimLogic
VAR_INPUT
END_VAR
(* No error or substitude values in sim mode *)
	stHstData.bError 	:= FALSE;
	stHstData.bSubsOn	:= FALSE;

(* Send data *)
	stStatus.nSendBoolData.0 		:= stDevData.bSend00;
	stStatus.nSendBoolData.1 		:= stDevData.bSend01;
	stStatus.nSendBoolData.2 		:= stDevData.bSend02;
	stStatus.nSendBoolData.3 		:= stDevData.bSend03;
	stStatus.nSendBoolData.4 		:= stDevData.bSend04;
	stStatus.nSendBoolData.5 		:= stDevData.bSend05;
	stStatus.nSendBoolData.6 		:= stDevData.bSend06;
	stStatus.nSendBoolData.7 		:= stDevData.bSend07;
	stStatus.nSendBoolData.8 		:= stDevData.bSend08;
	stStatus.nSendBoolData.9 		:= stDevData.bSend09;
	stStatus.nSendBoolData.10 		:= stDevData.bSend10;
	stStatus.nSendBoolData.11 		:= stDevData.bSend11;
	stStatus.nSendBoolData.12 		:= stDevData.bSend12;
	stStatus.nSendBoolData.13 		:= stDevData.bSend13;
	stStatus.nSendBoolData.14 		:= stDevData.bSend14;
	stStatus.nSendBoolData.15 		:= stDevData.bSend15;
	stStatus.nSendInt00				:= stDevData.nSend00;
	stStatus.nSendInt01				:= stDevData.nSend01;
	stStatus.nSendData				:= 16#80;
	stStatus.nSendSequenceNumber 	:= 16#FFFF;
	stStatus.nSendCrc 				:= F_CalcCrc16(ADR(stStatus), 8, stConfig.nDpDpId, POLYNOM);
END_METHOD

END_FUNCTION_BLOCK

// ---- Common/ProfidriveParamInterpreter/FB_ProfidriveParamInterpreter.TcPOU
FUNCTION_BLOCK PUBLIC FB_ProfidriveParamInterpreter
VAR_INPUT
	(* Pointer to raw user data *)
	pRawData		: POINTER TO BYTE;
	(* Pointer to array of parameters *)
	pParamSet		: POINTER TO ST_ProfidriveParam_Set;
END_VAR
VAR_OUTPUT
	(* Reference number for response *)
	nReference		: BYTE;
	(* 1 = read, 2 = write *)
	nCommand		: BYTE;
	(* Addressed axis number *)
	nAxis			: BYTE;
	(* Number of parameters to read/write *)
	nParameters		: BYTE;
END_VAR
VAR
	nOffsReq		: BYTE;
	nOffsValue		: BYTE;
	nFormatSize		: BYTE;
	nValues			: BYTE;
	i, j, k			: UINT;
END_VAR

(* Copy header (first 4 bytes) *)
	nReference := pRawData[0];
	nCommand := pRawData[1];
	nAxis := pRawData[2];
	nParameters := pRawData[3];

(* Set request offset behind header *)
	nOffsReq := 4;

(* Set value offset behind last request *)
	nOffsValue := 4 + nParameters * 6;

(* Reset all parameters *)
	memset(pParamSet, 0, SIZEOF(ST_ProfidriveParam_Set));

(* Check parameter number *)	
	IF nParameters = 0 THEN
		RETURN;
	END_IF

(* Loop through number of parameter requests *)
	FOR i := 0 TO nParameters - 1 BY 1 DO
		
		(* Get parameter request information (6 bytes)... *)
		pParamSet^[i].nAttribute := pRawData[nOffsReq];
		pParamSet^[i].nElements := pRawData[nOffsReq + 1];
		pParamSet^[i].nNumber := pRawData[nOffsReq + 2] * 16#100 + pRawData[nOffsReq + 3];
		pParamSet^[i].nSubIndex := pRawData[nOffsReq + 4] * 16#100 + pRawData[nOffsReq + 5];
		
		(* ... and set offset to next request *)
		nOffsReq := nOffsReq + 6;
				
		(* Write command -> get values *)
		IF nCommand = 2 THEN		
			(* Get format *)
			nFormatSize := FormatSize(pRawData[nOffsValue]);
			pParamSet^[i].nFormat := FormatType(pRawData[nOffsValue]);
			nOffsValue := nOffsValue + 1;
			
			(* Get number of values *)
			nValues := pRawData[nOffsValue];
			nOffsValue := nOffsValue + 1;
			
			(* Loop through number of values *)
			FOR j := 0 TO nValues - 1 BY 1 DO
				
				(* Set value offset behind current values *)
				nOffsValue := nOffsValue + nFormatSize;
				
				(* Loop through format size and get values in reverse order *)
				FOR k := 0 TO nFormatSize - 1 BY 1 DO
					pParamSet^[i].aValue[j + k] := pRawData[nOffsValue - k - 1];
				END_FOR
			END_FOR
			
			(* Check if odd and set to even number *)
			IF nOffsValue.0 THEN
				nOffsValue := nOffsValue + 1;
			END_IF
		END_IF
	END_FOR

METHOD INTERNAL FormatSize : BYTE
VAR_INPUT
	nFormat	: BYTE;
END_VAR
CASE nFormat OF
	 16#02 : FormatSize := 2;
	 16#03 : FormatSize := 2;
	 16#04 : FormatSize := 4;
	 16#05 : FormatSize := 2;
	 16#06 : FormatSize := 2;
	 16#07 : FormatSize := 4;
	 16#08 : FormatSize := 4;
	 16#40 : FormatSize := 0;
	 16#41 : FormatSize := 2;
	 16#42 : FormatSize := 2;
	 16#43 : FormatSize := 4;
	 16#44 : FormatSize := 0;
ELSE
	FormatSize := 0;
END_CASE
END_METHOD

METHOD INTERNAL FormatType : E_ProfidriveParam_Format
VAR_INPUT
	nFormat	: BYTE;
END_VAR
CASE nFormat OF
	 16#02 : FormatType := E_ProfidriveParam_Format.INT8;
	 16#03 : FormatType := E_ProfidriveParam_Format.INT16;
	 16#04 : FormatType := E_ProfidriveParam_Format.INT32;
	 16#05 : FormatType := E_ProfidriveParam_Format.UINT8;
	 16#06 : FormatType := E_ProfidriveParam_Format.UINT16;
	 16#07 : FormatType := E_ProfidriveParam_Format.UINT32;
	 16#08 : FormatType := E_ProfidriveParam_Format.FLOAT;
	 16#40 : FormatType := E_ProfidriveParam_Format.ZERO;
	 16#41 : FormatType := E_ProfidriveParam_Format.BYTE_;
	 16#42 : FormatType := E_ProfidriveParam_Format.WORD_;
	 16#43 : FormatType := E_ProfidriveParam_Format.DWORD_;
	 16#44 : FormatType := E_ProfidriveParam_Format.ERROR;
ELSE
	FormatType := E_ProfidriveParam_Format.UNKNOWN;
END_CASE
END_METHOD

METHOD INTERNAL MakeResponse : BOOL
VAR_INPUT
	(* Pointer to acyclic user data *)
	pResData		: POINTER TO BYTE;
END_VAR
VAR
	nOffset			: BYTE;
	nFormatSize		: BYTE;
	i, j, k			: UINT;
END_VAR
(* Copy header (first 4 bytes) *)
	pResData[0] := nReference;
	pResData[1] := nCommand;
	pResData[2] := nAxis;
	pResData[3] := nParameters;

(* Set offset behind header *)
	nOffset := 4;
	
(* Check parameter number *)	
	IF nParameters = 0 THEN
		RETURN;
	END_IF

(* Loop through number of parameter requests *)
	FOR i := 0 TO nParameters - 1 BY 1 DO
		
		(* Set format *)
		pResData[nOffset] := pParamSet^[i].nFormat;
		nFormatSize := FormatSize(pParamSet^[i].nFormat);
		nOffset := nOffset + 1;
		
		(* Set number of values *)
		pResData[nOffset] := pParamSet^[i].nElements;
		nOffset := nOffset + 1;
		
		(* Loop through number of elements *)
		FOR j := 0 TO pParamSet^[i].nElements - 1 BY 1 DO
			
			(* Set value offset behind current values *)
			nOffset := nOffset + nFormatSize;
			
			(* Loop through format size and get values in reverse order *)
			
			IF nFormatSize > 0 THEN
				FOR k := 0 TO nFormatSize - 1 BY 1 DO
					pResData[nOffset - k - 1] := pParamSet^[i].aValue[j + k] ;
				END_FOR
			END_IF
			
		END_FOR
		
		(* Check if odd and set to even number *)
		IF nOffset.0 THEN
			nOffset := nOffset + 1;
		END_IF	
	END_FOR

(* Return true when finished *)
	MakeResponse := TRUE;
END_METHOD

METHOD INTERNAL Reset : BOOL
nReference := 0;
nCommand := 0;
nAxis := 0;
nParameters := 0;
memset(pParamSet, 0, SIZEOF(ST_ProfidriveParam_Set));
END_METHOD

END_FUNCTION_BLOCK

// ---- _backlog/Danfoss_VLT_MCA_120/FB_Danfoss_VLT_MCA_120.TcPOU
{attribute 'reflection'} 
(* The VLT® PROFINET MCA 120 is used in combination with:
• VLT® HVAC Drive FC 102
• VLT® Refrigeration Drive FC 103
• VLT® AQUA Drive FC 202
• VLT® AutomationDrive FC 301/302
• VLT® Decentral Drive FCD 302
 *)
FUNCTION_BLOCK FB_Danfoss_VLT_MCA_120 EXTENDS FB_LinkDataReal
VAR_INPUT	
	stControl				: ST_Danfoss_VLT_MCA_120_Control;	
	stConfig 				: ST_Danfoss_VLT_MCA_120_Config;
END_VAR

VAR_OUTPUT
	stStatus				: ST_Danfoss_VLT_MCA_120_Status;
	fValue					: REAL;
END_VAR

VAR
    {attribute 'instance-path'} 
    {attribute 'noinit'} 
    sPath 					: STRING; 
	pFromBus				: POINTER TO BYTE;
	pToBus					: POINTER TO BYTE;	
	                    	
	fbProfidriveGSM			: FB_ProfidriveGSM;	
	fbMoveVelocity			: FB_MoveVelocity;
	
	fAcceleration	 		: REAL;
	fDeceleration		 	: REAL;
	fDecelerationQuickStop 	: REAL;
	fDecelerationCoastStop 	: REAL;
	bQuickStopExternal		: BOOL;
	
	bFaultPresent 			: BOOL;
	bAlarmPresent 			: BOOL;
	bInverterError 			: BOOL;
	bVoltageError 			: BOOL;
	bMomentError 			: BOOL;
	bTimerError 			: BOOL;
END_VAR

SUPER^();
InitRun();
ReadBus();
ControlLogic();
WriteBus();

(*Assign Process Data Objects to device*)
METHOD PUBLIC AssignProcessData : BOOL
VAR_INPUT
	aControlData 		: ANY; //Addr. Process Output (PO), 6 BYTES FROM FIELDBUS
	aStatusData 		: ANY; //Addr. Process Input (PI), 6 BYTES TO FIELDBUS
END_VAR
THIS^.pFromBus := aControlData.pValue;
THIS^.pToBus := aStatusData.pValue;
END_METHOD

METHOD INTERNAL ControlLogic
(* Evaluate/limit parameters *)
	EvaluateParameters();

(* Unity init - load position *)
	IF SUPER^.Status.7 THEN
		ControlData := StatusData;
	END_IF

(* Call base statemachine *)
fbProfidriveGSM.bStandstill						:= OC_Core.F_Compare(fbMoveVelocity.fVelocity, 0, 1E-3);
fbProfidriveGSM.stControl.b0_On 				:= stControl.bOFF1;
fbProfidriveGSM.stControl.b1_CoastStop 			:= stControl.bOFF2;
fbProfidriveGSM.stControl.b2_QuickStop 			:= stControl.bOFF3 AND NOT bQuickStopExternal;
fbProfidriveGSM.stControl.b3_EnableOperation	:= stControl.bEnableOperation;

(* Preset target values *)
	fbMoveVelocity.fTargetVelocity	:= 0;
	fbMoveVelocity.fAccMax 			:= fAcceleration;
	fbMoveVelocity.fDecMax 			:= fDeceleration;

(* Operation *)
	IF fbProfidriveGSM.eState = E_ProfidriveGSM_State.S4_Operation THEN	
		// Main setpoint
		IF NOT stControl.bJog1 AND NOT stControl.bJog2 THEN
			fbMoveVelocity.fTargetVelocity := (stControl.nSoll * stConfig.fP2000) / 16#4000;
		// Jog 1
		ELSIF stControl.bJog1 AND NOT stControl.bJog2 THEN
			fbMoveVelocity.fTargetVelocity := stConfig.fP1058;
		// Jog 2
		ELSIF NOT stControl.bJog1 AND stControl.bJog2 THEN	
			fbMoveVelocity.fTargetVelocity := stConfig.fP1059;
		END_IF
		
		// Stop
		IF NOT stControl.bOperatingCondition OR NOT stControl.bEnableSetpoint THEN
			fbMoveVelocity.fTargetVelocity := 0;
		END_IF
		
		// Reversing velocity
		IF stControl.bReversing THEN
			fbMoveVelocity.fTargetVelocity := -fbMoveVelocity.fTargetVelocity;
		END_IF
		
		// Hold velocity
		IF NOT stControl.bContinueRampFunctionGenerator AND NOT stControl.bJog1 AND NOT stControl.bJog2 THEN
			fbMoveVelocity.fTargetVelocity := fbMoveVelocity.fVelocity;
		END_IF	
		
	END_IF
	
